KUKA KRL program: MyProgram_041().src

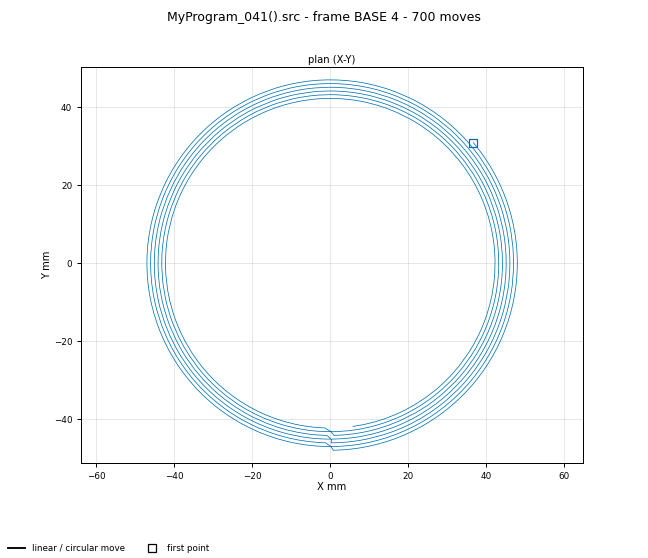
[picture p0: tool path of MyProgram_041().src in frame BASE 4, 700 of 700 moves have a stored position in this frame; points joined in program order, loops and branches not executed]
&ACCESS RVP
&REL 1
&PARAM TEMPLATE = C:\KRC\Roboter\Template\vorgabe
&PARAM EDITMASK = *
DEF MyProgram_041()
; ---- Setting reference (Base) ----
$BASE = BASE_DATA[4]

; --------------------------
; ---- Setting tool (TCP) ----
$TOOL = TOOL_DATA[3]
; --------------------------

$VEL.CP = VEL_APROX_PRINT
Startdeposition()
$VEL.CP = VEL_PRINT
LIN {X 36.6763,Y 30.8604,Z 63,A 32.6646,B 24.8495,C -2.8306,E1 25.1236,E2 -309.1779} C_DIS
LIN {X 38.1464,Y 29.0236,Z 63,A 29.8672,B 24.8502,C -2.8243,E1 25.1284,E2 -306.3787} C_DIS
LIN {X 39.5245,Y 27.1169,Z 63,A 27.0703,B 24.8509,C -2.8177,E1 25.1329,E2 -303.5798} C_DIS
LIN {X 40.8075,Y 25.1448,Z 63,A 24.2742,B 24.8516,C -2.8108,E1 25.1371,E2 -300.7815} C_DIS
LIN {X 41.9921,Y 23.1122,Z 63,A 21.4787,B 24.8523,C -2.8037,E1 25.141,E2 -297.9837} C_DIS
LIN {X 43.0756,Y 21.0239,Z 63,A 18.6835,B 24.8531,C -2.7964,E1 25.1445,E2 -295.1861} C_DIS
LIN {X 44.0553,Y 18.885,Z 63,A 15.8888,B 24.8539,C -2.7889,E1 25.1476,E2 -292.389} C_DIS
LIN {X 44.9289,Y 16.7005,Z 63,A 13.0946,B 24.8547,C -2.7812,E1 25.1505,E2 -289.5921} C_DIS
LIN {X 45.6942,Y 14.4759,Z 63,A 10.3007,B 24.8555,C -2.7734,E1 25.1529,E2 -286.7955} C_DIS
LIN {X 46.3495,Y 12.2163,Z 63,A 7.5073,B 24.8564,C -2.7654,E1 25.155,E2 -283.9992} C_DIS
LIN {X 46.8931,Y 9.9273,Z 63,A 4.7141,B 24.8572,C -2.7573,E1 25.1567,E2 -281.203} C_DIS
LIN {X 47.3237,Y 7.6144,Z 63,A 1.9212,B 24.8581,C -2.749,E1 25.158,E2 -278.4069} C_DIS
LIN {X 47.6194,Y 5.4623,Z 63,A -0.6575,B 24.8589,C -2.7414,E1 25.1589,E2 -275.8254} C_DIS
LIN {X 47.83,Y 3.1192,Z 63,A -3.4502,B 24.8597,C -2.733,E1 25.1596,E2 -273.0294} C_DIS
LIN {X 47.9255,Y 0.7685,Z 63,A -6.2425,B 24.8606,C -2.7246,E1 25.1598,E2 -270.2338} C_DIS
LIN {X 47.9207,Y -1.0254,Z 63,A -8.406,B 24.8613,C -2.7174,E1 25.1597,E2 -268.0664} C_DIS
LIN {X 47.8025,Y -3.5261,Z 63,A -11.3432,B 24.8622,C -2.7091,E1 25.1592,E2 -265.1268} C_DIS
LIN {X 47.5719,Y -5.8674,Z 63,A -14.1356,B 24.863,C -2.7006,E1 25.1583,E2 -262.3309} C_DIS
LIN {X 47.2267,Y -8.1946,Z 63,A -16.9281,B 24.8639,C -2.6922,E1 25.1571,E2 -259.5348} C_DIS
LIN {X 46.7677,Y -10.502,Z 63,A -19.7204,B 24.8647,C -2.6838,E1 25.1555,E2 -256.7389} C_DIS
LIN {X 46.1961,Y -12.7842,Z 63,A -22.5132,B 24.8656,C -2.6755,E1 25.1535,E2 -253.9426} C_DIS
LIN {X 45.5132,Y -15.0355,Z 63,A -25.3061,B 24.8664,C -2.6672,E1 25.1511,E2 -251.146} C_DIS
LIN {X 44.7206,Y -17.2506,Z 63,A -28.0993,B 24.8672,C -2.6591,E1 25.1484,E2 -248.3492} C_DIS
LIN {X 43.8203,Y -19.4242,Z 63,A -30.8927,B 24.868,C -2.6511,E1 25.1454,E2 -245.5521} C_DIS
LIN {X 42.8144,Y -21.5509,Z 63,A -33.6867,B 24.8688,C -2.6432,E1 25.1419,E2 -242.7545} C_DIS
LIN {X 41.7053,Y -23.6258,Z 63,A -36.4807,B 24.8696,C -2.6355,E1 25.1382,E2 -239.957} C_DIS
LIN {X 40.4959,Y -25.6437,Z 63,A -39.2754,B 24.8703,C -2.628,E1 25.1341,E2 -237.1587} C_DIS
LIN {X 39.1888,Y -27.5999,Z 63,A -42.0705,B 24.871,C -2.6207,E1 25.1296,E2 -234.36} C_DIS
LIN {X 37.7873,Y -29.4895,Z 63,A -44.8661,B 24.8717,C -2.6136,E1 25.1249,E2 -231.5609} C_DIS
LIN {X 36.2948,Y -31.3081,Z 63,A -47.6623,B 24.8724,C -2.6067,E1 25.1199,E2 -228.7612} C_DIS
LIN {X 34.7149,Y -33.0513,Z 63,A -50.4591,B 24.8731,C -2.6001,E1 25.1146,E2 -225.961} C_DIS
LIN {X 32.9356,Y -34.8237,Z 63,A -53.4601,B 24.8738,C -2.5931,E1 25.1086,E2 -222.9559} C_DIS
LIN {X 31.0875,Y -36.4828,Z 63,A -56.467,B 24.8745,C -2.5857,E1 25.1022,E2 -219.9435} C_DIS
LIN {X 29.0236,Y -38.1464,Z 63,A -59.5531,B 24.875,C -2.5805,E1 25.0954,E2 -216.8565} C_DIS
LIN {X 27.1169,Y -39.5245,Z 63,A -62.3528,B 24.8755,C -2.5751,E1 25.089,E2 -214.0537} C_DIS
LIN {X 25.1448,Y -40.8075,Z 63,A -65.1533,B 24.876,C -2.5701,E1 25.0824,E2 -211.2502} C_DIS
LIN {X 23.1122,Y -41.9921,Z 63,A -67.9546,B 24.8765,C -2.5654,E1 25.0756,E2 -208.4461} C_DIS
LIN {X 21.0239,Y -43.0756,Z 63,A -70.7565,B 24.8769,C -2.561,E1 25.0686,E2 -205.6414} C_DIS
LIN {X 18.885,Y -44.0553,Z 63,A -73.5596,B 24.8773,C -2.557,E1 25.0615,E2 -202.8357} C_DIS
LIN {X 16.7005,Y -44.9289,Z 63,A -76.3635,B 24.8776,C -2.5534,E1 25.0542,E2 -200.0294} C_DIS
LIN {X 14.4759,Y -45.6942,Z 63,A -79.1682,B 24.8779,C -2.5501,E1 25.0467,E2 -197.2223} C_DIS
LIN {X 12.2163,Y -46.3495,Z 63,A -81.9739,B 24.8782,C -2.5472,E1 25.0392,E2 -194.4144} C_DIS
LIN {X 9.9273,Y -46.8931,Z 63,A -84.7806,B 24.8784,C -2.5448,E1 25.0315,E2 -191.6057} C_DIS
LIN {X 7.6145,Y -47.3237,Z 63,A -87.5882,B 24.8786,C -2.5427,E1 25.0238,E2 -188.7961} C_DIS
LIN {X 5.4623,Y -47.6194,Z 63,A -90.0984,B 24.8786,C -2.5426,E1 25.0168,E2 -186.2875} C_DIS
LIN {X 3.1192,Y -47.83,Z 63,A -92.991,B 24.8789,C -2.5399,E1 25.0088,E2 -183.3901} C_DIS
LIN {X 0.7685,Y -47.9255,Z 63,A -95.7979,B 24.8789,C -2.5391,E1 25.0009,E2 -180.5818} C_DIS
LIN {X 0.7685,Y -47.9255,Z 63,A -95.7979,B 24.8789,C -2.5391,E1 25.0009,E2 -180.5818} C_DIS
Enddeposition()
LIN {X 0.2143,Y -46.9784,Z 63,A -95.4397,B 24.8758,C -2.5723,E1 25.0021,E2 -181.019} C_DIS
Startdeposition()
$VEL.CP = VEL_PRINT
LIN {X 2.5559,Y -46.9121,Z 63,A -92.1955,B 24.8751,C -2.5797,E1 25.0112,E2 -184.2799} C_DIS
LIN {X 5.1846,Y -46.6955,Z 63,A -89.0891,B 24.8751,C -2.5796,E1 25.0199,E2 -187.3841} C_DIS
LIN {X 7.4092,Y -46.3943,Z 63,A -86.2366,B 24.8747,C -2.5834,E1 25.0278,E2 -190.2431} C_DIS
LIN {X 9.682,Y -45.9738,Z 63,A -83.5774,B 24.8747,C -2.583,E1 25.035,E2 -192.8981} C_DIS
LIN {X 12.0789,Y -45.4027,Z 63,A -80.419,B 24.8742,C -2.5887,E1 25.0436,E2 -196.0652} C_DIS
LIN {X 14.5681,Y -44.6661,Z 63,A -77.3449,B 24.874,C -2.5907,E1 25.0518,E2 -199.1385} C_DIS
LIN {X 16.8661,Y -43.8505,Z 63,A -74.3809,B 24.8736,C -2.5944,E1 25.0596,E2 -202.105} C_DIS
LIN {X 19.0655,Y -42.94,Z 63,A -71.3711,B 24.873,C -2.6005,E1 25.0673,E2 -205.1221} C_DIS
LIN {X 21.5139,Y -41.7666,Z 63,A -68.1734,B 24.8727,C -2.6038,E1 25.0753,E2 -208.319} C_DIS
LIN {X 23.5958,Y -40.6271,Z 63,A -65.3023,B 24.8723,C -2.6084,E1 25.0823,E2 -211.1926} C_DIS
LIN {X 25.6235,Y -39.3801,Z 63,A -62.7798,B 24.8724,C -2.6069,E1 25.0882,E2 -213.7033} C_DIS
LIN {X 27.3032,Y -38.2334,Z 63,A -59.8844,B 24.8712,C -2.6194,E1 25.0949,E2 -216.6186} C_DIS
LIN {X 29.4691,Y -36.5899,Z 63,A -56.4143,B 24.8702,C -2.6293,E1 25.1026,E2 -220.0991} C_DIS
LIN {X 31.6335,Y -34.7366,Z 63,A -52.8319,B 24.8692,C -2.6391,E1 25.1101,E2 -223.6906} C_DIS
LIN {X 33.711,Y -32.7242,Z 63,A -49.5665,B 24.8689,C -2.6426,E1 25.1165,E2 -226.9504} C_DIS
LIN {X 35.4262,Y -30.8588,Z 63,A -46.5387,B 24.8682,C -2.6491,E1 25.1221,E2 -229.9802} C_DIS
LIN {X 36.9362,Y -29.0346,Z 63,A -43.7525,B 24.8677,C -2.6547,E1 25.127,E2 -232.7665} C_DIS
LIN {X 38.153,Y -27.4162,Z 63,A -41.5295,B 24.8675,C -2.6566,E1 25.1307,E2 -234.9833} C_DIS
LIN {X 39.4006,Y -25.5917,Z 63,A -38.491,B 24.8661,C -2.6705,E1 25.1354,E2 -238.0396} C_DIS
LIN {X 40.6723,Y -23.5171,Z 63,A -35.6061,B 24.8654,C -2.6773,E1 25.1395,E2 -240.9257} C_DIS
LIN {X 41.8533,Y -21.3443,Z 63,A -32.6333,B 24.8646,C -2.6851,E1 25.1434,E2 -243.9014} C_DIS
LIN {X 42.6017,Y -19.8084,Z 63,A -30.3873,B 24.8637,C -2.6944,E1 25.146,E2 -246.1573} C_DIS
LIN {X 43.7378,Y -17.1547,Z 63,A -27.0571,B 24.863,C -2.7012,E1 25.1496,E2 -249.4853} C_DIS
LIN {X 44.6118,Y -14.7336,Z 63,A -23.7996,B 24.8618,C -2.7131,E1 25.1525,E2 -252.7525} C_DIS
LIN {X 45.4336,Y -11.9641,Z 63,A -20.8446,B 24.8618,C -2.7129,E1 25.1548,E2 -255.6901} C_DIS
LIN {X 46.1112,Y -9.0029,Z 63,A -15.9869,B 24.8583,C -2.747,E1 25.1576,E2 -260.6001} C_DIS
LIN {X 46.6067,Y -5.9251,Z 63,A -12.4483,B 24.8576,C -2.7537,E1 25.1589,E2 -264.1337} C_DIS
LIN {X 46.9567,Y -1.5325,Z 63,A -7.5964,B 24.8569,C -2.7604,E1 25.1598,E2 -268.9726} C_DIS
LIN {X 46.9771,Y 0.6801,Z 63,A -4.6126,B 24.8554,C -2.7744,E1 25.1597,E2 -271.9719} C_DIS
LIN {X 46.8023,Y 4.1062,Z 63,A -0.522,B 24.8542,C -2.7856,E1 25.1589,E2 -276.0648} C_DIS
LIN {X 46.3299,Y 7.7988,Z 63,A 3.3596,B 24.8542,C -2.7869,E1 25.1574,E2 -279.9263} C_DIS
LIN {X 45.9041,Y 10.0043,Z 63,A 6.6583,B 24.8521,C -2.806,E1 25.1555,E2 -283.251} C_DIS
LIN {X 45.2529,Y 12.6287,Z 63,A 9.5452,B 24.8519,C -2.8079,E1 25.1534,E2 -286.1258} C_DIS
LIN {X 44.6509,Y 14.615,Z 63,A 12.1852,B 24.8509,C -2.8174,E1 25.1512,E2 -288.7733} C_DIS
LIN {X 43.8399,Y 16.8942,Z 63,A 15.8973,B 24.8484,C -2.8405,E1 25.1475,E2 -292.5194} C_DIS
LIN {X 42.3575,Y 20.3254,Z 63,A 19.7008,B 24.8486,C -2.8387,E1 25.1431,E2 -296.298} C_DIS
LIN {X 41.1665,Y 22.6422,Z 63,A 22.7618,B 24.8479,C -2.8449,E1 25.1391,E2 -299.3577} C_DIS
LIN {X 40.0354,Y 24.5864,Z 63,A 25.8315,B 24.8465,C -2.8582,E1 25.1347,E2 -302.4431} C_DIS
LIN {X 38.3506,Y 27.1393,Z 63,A 29.1136,B 24.8465,C -2.859,E1 25.1295,E2 -305.7111} C_DIS
LIN {X 37.1165,Y 28.8039,Z 63,A 31.388,B 24.8463,C -2.8604,E1 25.1257,E2 -307.9778} C_DIS
LIN {X 35.589,Y 30.672,Z 63,A 34.6406,B 24.8449,C -2.8728,E1 25.1199,E2 -311.2449} C_DIS
LIN {X 34.078,Y 32.3421,Z 63,A 37.4842,B 24.8441,C -2.8805,E1 25.1145,E2 -314.0943} C_DIS
LIN {X 32.1994,Y 34.2122,Z 63,A 40.6791,B 24.8435,C -2.8864,E1 25.108,E2 -317.2899} C_DIS
LIN {X 30.3202,Y 35.8887,Z 63,A 43.688,B 24.8429,C -2.8911,E1 25.1017,E2 -320.2982} C_DIS
LIN {X 28.4537,Y 37.3863,Z 63,A 46.7319,B 24.8421,C -2.8986,E1 25.095,E2 -323.3484} C_DIS
LIN {X 26.3,Y 38.9303,Z 63,A 49.9644,B 24.8416,C -2.9038,E1 25.0876,E2 -326.5823} C_DIS
LIN {X 23.9042,Y 40.4458,Z 63,A 53.0971,B 24.8416,C -2.9032,E1 25.0801,E2 -329.7037} C_DIS
LIN {X 21.9009,Y 41.5647,Z 63,A 56.1163,B 24.8408,C -2.9108,E1 25.0727,E2 -332.7322} C_DIS
LIN {X 20.3598,Y 42.3409,Z 63,A 58.9872,B 24.8391,C -2.9266,E1 25.0654,E2 -335.6331} C_DIS
LIN {X 16.672,Y 43.924,Z 63,A 63.0887,B 24.84,C -2.9178,E1 25.0549,E2 -339.7044} C_DIS
LIN {X 14.163,Y 44.7968,Z 63,A 66.3896,B 24.8396,C -2.9214,E1 25.0461,E2 -343.0076} C_DIS
LIN {X 11.5862,Y 45.5307,Z 63,A 69.5926,B 24.8396,C -2.9224,E1 25.0375,E2 -346.2078} C_DIS
LIN {X 8.9483,Y 46.1217,Z 63,A 72.8147,B 24.8395,C -2.9226,E1 25.0287,E2 -349.4264} C_DIS
LIN {X 7.0373,Y 46.4518,Z 63,A 75.1648,B 24.8395,C -2.9231,E1 25.0222,E2 -351.7753} C_DIS
LIN {X 4.6739,Y 46.7491,Z 63,A 78.1637,B 24.8392,C -2.9251,E1 25.0139,E2 -354.7767} C_DIS
LIN {X 2.015,Y 46.9384,Z 63,A 81.4087,B 24.8392,C -2.9249,E1 25.0048,E2 -358.0203} C_DIS
LIN {X -0.6275,Y 46.9781,Z 63,A 84.1397,B 24.8402,C -2.9165,E1 24.9973,E2 -360.7311} C_DIS
LIN {X -2.9749,Y 46.8878,Z 63,A 87.5384,B 24.8393,C -2.9239,E1 24.9877,E2 -364.1482} C_DIS
LIN {X -5.5799,Y 46.6493,Z 63,A 90.7209,B 24.8395,C -2.9221,E1 24.9789,E2 -367.3283} C_DIS
LIN {X -7.976,Y 46.3002,Z 63,A 93.578,B 24.8399,C -2.9186,E1 24.971,E2 -370.1797} C_DIS
LIN {X -10.1804,Y 45.8657,Z 63,A 96.0614,B 24.8406,C -2.9125,E1 24.9643,E2 -372.6513} C_DIS
LIN {X -12.438,Y 45.3057,Z 63,A 99.2139,B 24.8404,C -2.9144,E1 24.9557,E2 -375.8132} C_DIS
LIN {X -14.0781,Y 44.8231,Z 63,A 102.2726,B 24.839,C -2.9267,E1 24.9475,E2 -378.9066} C_DIS
LIN {X -17.8756,Y 43.4484,Z 63,A 106.2167,B 24.8414,C -2.9057,E1 24.9373,E2 -382.8088} C_DIS
LIN {X -20.1909,Y 42.4221,Z 63,A 109.3156,B 24.8418,C -2.9012,E1 24.9295,E2 -385.9049} C_DIS
LIN {X -21.88,Y 41.5757,Z 63,A 112.0704,B 24.8415,C -2.904,E1 24.9226,E2 -388.6739} C_DIS
LIN {X -24.7808,Y 39.915,Z 63,A 115.744,B 24.843,C -2.891,E1 24.9139,E2 -392.3276} C_DIS
LIN {X -26.8595,Y 38.5467,Z 63,A 118.8267,B 24.8435,C -2.8858,E1 24.9068,E2 -395.4084} C_DIS
LIN {X -29.0273,Y 36.9419,Z 63,A 122.1517,B 24.8442,C -2.8796,E1 24.8994,E2 -398.7304} C_DIS
LIN {X -31.0833,Y 35.2301,Z 63,A 124.9609,B 24.8457,C -2.8662,E1 24.8935,E2 -401.5186} C_DIS
LIN {X -32.2942,Y 34.123,Z 63,A 127.5606,B 24.8453,C -2.8698,E1 24.8881,E2 -404.1375} C_DIS
LIN {X -34.3301,Y 32.074,Z 63,A 130.986,B 24.8463,C -2.8601,E1 24.8815,E2 -407.5544} C_DIS
LIN {X -36.1116,Y 30.0538,Z 63,A 134.2654,B 24.8472,C -2.8518,E1 24.8755,E2 -410.8289} C_DIS
LIN {X -37.7375,Y 27.9862,Z 63,A 137.0526,B 24.8487,C -2.8378,E1 24.8708,E2 -413.5958} C_DIS
LIN {X -38.8546,Y 26.4122,Z 63,A 139.9102,B 24.8487,C -2.8382,E1 24.8663,E2 -416.4685} C_DIS
LIN {X -40.3999,Y 23.982,Z 63,A 143.4333,B 24.8497,C -2.8286,E1 24.8611,E2 -419.9866} C_DIS
LIN {X -41.7299,Y 21.5857,Z 63,A 146.753,B 24.8507,C -2.8187,E1 24.8567,E2 -423.3003} C_DIS
LIN {X -42.7838,Y 19.4124,Z 63,A 149.9969,B 24.8512,C -2.814,E1 24.8529,E2 -426.5507} C_DIS
LIN {X -44.1351,Y 16.1049,Z 63,A 154.0955,B 24.853,C -2.7976,E1 24.8488,E2 -430.633} C_DIS
LIN {X -44.8607,Y 13.9568,Z 63,A 156.6924,B 24.8541,C -2.787,E1 24.8466,E2 -433.2194} C_DIS
LIN {X -45.5111,Y 11.6624,Z 63,A 159.7162,B 24.8549,C -2.7795,E1 24.8443,E2 -436.2429} C_DIS
LIN {X -46.0396,Y 9.3616,Z 63,A 162.7323,B 24.8556,C -2.7723,E1 24.8426,E2 -439.2596} C_DIS
LIN {X -46.4956,Y 6.7422,Z 63,A 165.7745,B 24.857,C -2.7596,E1 24.8412,E2 -442.2894} C_DIS
LIN {X -46.7606,Y 4.558,Z 63,A 168.776,B 24.8574,C -2.7553,E1 24.8403,E2 -445.2986} C_DIS
LIN {X -46.9449,Y 1.8632,Z 63,A 171.9898,B 24.8586,C -2.7439,E1 24.8398,E2 -448.5045} C_DIS
LIN {X -46.9769,Y -0.6903,Z 63,A 175.163,B 24.8595,C -2.7349,E1 24.8398,E2 -451.6753} C_DIS
LIN {X -46.8667,Y -3.2866,Z 63,A 178.2443,B 24.8607,C -2.7239,E1 24.8403,E2 -454.7488} C_DIS
LIN {X -46.6945,Y -5.1937,Z 63,A -179.2053,B 24.8611,C -2.7194,E1 24.8411,E2 -457.3038} C_DIS
LIN {X -46.3138,Y -7.8948,Z 63,A -175.9746,B 24.8623,C -2.708,E1 24.8425,E2 -460.5264} C_DIS
LIN {X -45.8138,Y -10.4116,Z 63,A -172.7879,B 24.8632,C -2.6993,E1 24.8443,E2 -463.711} C_DIS
LIN {X -45.1647,Y -12.9399,Z 63,A -169.5411,B 24.864,C -2.6907,E1 24.8467,E2 -466.9561} C_DIS
LIN {X -44.3842,Y -15.4059,Z 63,A -166.7067,B 24.8654,C -2.6773,E1 24.8492,E2 -469.7745} C_DIS
LIN {X -43.6542,Y -17.3676,Z 63,A -163.9593,B 24.8659,C -2.6726,E1 24.8519,E2 -472.5262} C_DIS
LIN {X -42.5994,Y -19.8133,Z 63,A -160.4602,B 24.8664,C -2.6669,E1 24.8559,E2 -476.031} C_DIS
LIN {X -41.346,Y -22.3113,Z 63,A -157.1221,B 24.8675,C -2.6568,E1 24.8602,E2 -479.3628} C_DIS
LIN {X -40.0037,Y -24.6386,Z 63,A -153.944,B 24.8684,C -2.647,E1 24.8647,E2 -482.5338} C_DIS
LIN {X -38.8415,Y -26.4316,Z 63,A -151.505,B 24.8693,C -2.6382,E1 24.8685,E2 -484.9641} C_DIS
LIN {X -37.5666,Y -28.2139,Z 63,A -148.5222,B 24.8695,C -2.6361,E1 24.8734,E2 -487.9563} C_DIS
LIN {X -35.9165,Y -30.2876,Z 63,A -145.3045,B 24.8703,C -2.6285,E1 24.8791,E2 -491.1707} C_DIS
LIN {X -34.1655,Y -32.249,Z 63,A -142.6079,B 24.8717,C -2.6144,E1 24.8842,E2 -493.8456} C_DIS
LIN {X -32.5987,Y -33.832,Z 63,A -139.3792,B 24.8715,C -2.6161,E1 24.8906,E2 -497.0918} C_DIS
LIN {X -30.6979,Y -35.5667,Z 63,A -136.1305,B 24.8719,C -2.6116,E1 24.8974,E2 -500.3429} C_DIS
LIN {X -29.145,Y -36.8489,Z 63,A -133.9522,B 24.8728,C -2.6032,E1 24.9021,E2 -502.5092} C_DIS
LIN {X -27.314,Y -38.2259,Z 63,A -130.9734,B 24.873,C -2.6012,E1 24.9088,E2 -505.4939} C_DIS
LIN {X -25.1237,Y -39.6996,Z 63,A -127.4866,B 24.873,C -2.6003,E1 24.917,E2 -508.9897} C_DIS
LIN {X -22.9515,Y -40.994,Z 63,A -124.3564,B 24.8734,C -2.5968,E1 24.9246,E2 -512.1208} C_DIS
LIN {X -20.2336,Y -42.4016,Z 63,A -120.8547,B 24.8742,C -2.5888,E1 24.9333,E2 -515.6127} C_DIS
LIN {X -18.3269,Y -43.2598,Z 63,A -118.4196,B 24.8746,C -2.5844,E1 24.9395,E2 -518.043} C_DIS
LIN {X -16.0279,Y -44.1632,Z 63,A -115.2725,B 24.8746,C -2.5837,E1 24.9478,E2 -521.1952} C_DIS
LIN {X -13.4838,Y -45.0053,Z 63,A -111.9643,B 24.8748,C -2.582,E1 24.9566,E2 -524.5051} C_DIS
LIN {X -10.8546,Y -45.7114,Z 63,A -108.855,B 24.8753,C -2.5768,E1 24.965,E2 -527.6066} C_DIS
LIN {X -8.6723,Y -46.1748,Z 63,A -106.0396,B 24.8753,C -2.5773,E1 24.9727,E2 -530.4262} C_DIS
LIN {X -6.3616,Y -46.5496,Z 63,A -103.1497,B 24.8753,C -2.5772,E1 24.9807,E2 -533.3183} C_DIS
LIN {X -3.8273,Y -46.8256,Z 63,A -99.9519,B 24.8752,C -2.5784,E1 24.9896,E2 -536.5206} C_DIS
LIN {X -1.3952,Y -46.961,Z 63,A -97.0343,B 24.8752,C -2.5778,E1 24.9977,E2 -539.4375} C_DIS
LIN {X 0.2143,Y -46.9784,Z 63,A -95.4395,B 24.8758,C -2.5722,E1 25.0021,E2 -541.019} C_DIS
Enddeposition()
LIN {X 0.2143,Y -46.9784,Z 63,A -95.4395,B 24.8758,C -2.5722,E1 25.0021,E2 -541.019} C_DIS
Startdeposition()
$VEL.CP = VEL_PRINT
LIN {X -1.2064,Y -46.0165,Z 63,A -98.1296,B 24.8757,C -2.5734,E1 24.9946,E2 -538.3316} C_DIS
LIN {X -2.996,Y -45.9343,Z 63,A -100.6273,B 24.8761,C -2.5691,E1 24.9876,E2 -535.823} C_DIS
LIN {X -5.5683,Y -45.6943,Z 63,A -103.8573,B 24.8761,C -2.5693,E1 24.9787,E2 -532.5914} C_DIS
LIN {X -8.1693,Y -45.3011,Z 63,A -107.3449,B 24.8763,C -2.567,E1 24.969,E2 -529.0951} C_DIS
LIN {X -10.6177,Y -44.7912,Z 63,A -110.1372,B 24.8757,C -2.5732,E1 24.9615,E2 -526.314} C_DIS
LIN {X -12.9468,Y -44.1739,Z 63,A -113.2311,B 24.8757,C -2.5737,E1 24.9531,E2 -523.2164} C_DIS
LIN {X -15.3538,Y -43.3959,Z 63,A -116.3054,B 24.8753,C -2.5773,E1 24.945,E2 -520.1448} C_DIS
LIN {X -18.1446,Y -42.3057,Z 63,A -119.8982,B 24.8748,C -2.5829,E1 24.9357,E2 -516.5574} C_DIS
LIN {X -19.9975,Y -41.4612,Z 63,A -122.8081,B 24.875,C -2.5804,E1 24.9283,E2 -513.6341} C_DIS
LIN {X -22.5947,Y -40.1054,Z 63,A -125.9036,B 24.8738,C -2.5929,E1 24.9208,E2 -510.5598} C_DIS
LIN {X -23.9436,Y -39.3146,Z 63,A -128.1392,B 24.8739,C -2.5916,E1 24.9154,E2 -508.3143} C_DIS
LIN {X -25.6481,Y -38.2249,Z 63,A -130.5652,B 24.8734,C -2.5967,E1 24.9097,E2 -505.8925} C_DIS
LIN {X -27.056,Y -37.2411,Z 63,A -133.252,B 24.8738,C -2.5926,E1 24.9036,E2 -503.1867} C_DIS
LIN {X -28.9064,Y -35.824,Z 63,A -135.8534,B 24.8729,C -2.6019,E1 24.8979,E2 -500.5977} C_DIS
LIN {X -30.8319,Y -34.1812,Z 63,A -138.9812,B 24.8723,C -2.6082,E1 24.8914,E2 -497.4727} C_DIS
LIN {X -33.3178,Y -31.7629,Z 63,A -142.8699,B 24.8708,C -2.6228,E1 24.8837,E2 -493.6024} C_DIS
LIN {X -35.1938,Y -29.6705,Z 63,A -146.9276,B 24.8708,C -2.6231,E1 24.8762,E2 -489.5271} C_DIS
LIN {X -36.5981,Y -27.9205,Z 63,A -149.5235,B 24.8699,C -2.6322,E1 24.8717,E2 -486.9408} C_DIS
LIN {X -38.1584,Y -25.7462,Z 63,A -152.927,B 24.8692,C -2.6394,E1 24.8663,E2 -483.5377} C_DIS
LIN {X -39.398,Y -23.8063,Z 63,A -155.8746,B 24.8686,C -2.6456,E1 24.8619,E2 -480.5899} C_DIS
LIN {X -40.6461,Y -21.6068,Z 63,A -159.8006,B 24.8687,C -2.6441,E1 24.8567,E2 -476.6397} C_DIS
LIN {X -41.8492,Y -19.1742,Z 63,A -163.1919,B 24.8678,C -2.6532,E1 24.8527,E2 -473.2516} C_DIS
LIN {X -43.1775,Y -15.9583,Z 63,A -166.9255,B 24.8658,C -2.673,E1 24.8489,E2 -469.5443} C_DIS
LIN {X -44.4043,Y -12.1328,Z 63,A -171.4229,B 24.8637,C -2.6939,E1 24.8453,E2 -465.0712} C_DIS
LIN {X -44.8415,Y -10.4003,Z 63,A -174.104,B 24.8637,C -2.6949,E1 24.8435,E2 -462.3767} C_DIS
LIN {X -45.347,Y -7.9143,Z 63,A -177.23,B 24.8626,C -2.7049,E1 24.8418,E2 -459.2561} C_DIS
LIN {X -45.7486,Y -5.1043,Z 63,A 178.9324,B 24.8619,C -2.7121,E1 24.8405,E2 -455.4127} C_DIS
LIN {X -45.971,Y -2.3719,Z 63,A 175.7437,B 24.8605,C -2.7254,E1 24.8399,E2 -452.2368} C_DIS
LIN {X -46.0317,Y 0.1331,Z 63,A 172.5788,B 24.8595,C -2.7346,E1 24.8398,E2 -449.0748} C_DIS
LIN {X -45.9564,Y 2.6362,Z 63,A 169.1185,B 24.859,C -2.7403,E1 24.8402,E2 -445.6072} C_DIS
LIN {X -45.6948,Y 5.5633,Z 63,A 165.7078,B 24.8575,C -2.7547,E1 24.8412,E2 -442.2107} C_DIS
LIN {X -45.3131,Y 8.1024,Z 63,A 162.5598,B 24.8564,C -2.7653,E1 24.8427,E2 -439.0693} C_DIS
LIN {X -44.8166,Y 10.5083,Z 63,A 159.1164,B 24.8559,C -2.7701,E1 24.8448,E2 -435.6172} C_DIS
LIN {X -43.7953,Y 14.1738,Z 63,A 154.9462,B 24.8536,C -2.7916,E1 24.848,E2 -431.4741} C_DIS
LIN {X -42.8735,Y 16.7571,Z 63,A 151.1618,B 24.853,C -2.7973,E1 24.8517,E2 -427.682} C_DIS
LIN {X -42.0147,Y 18.8062,Z 63,A 148.3926,B 24.8522,C -2.8054,E1 24.8548,E2 -424.917} C_DIS
LIN {X -40.6841,Y 21.5346,Z 63,A 144.617,B 24.851,C -2.8163,E1 24.8595,E2 -421.1473} C_DIS
LIN {X -39.3588,Y 23.8709,Z 63,A 141.6249,B 24.8495,C -2.8301,E1 24.8637,E2 -418.1726} C_DIS
LIN {X -38.6201,Y 25.0484,Z 63,A 139.4394,B 24.8496,C -2.8291,E1 24.867,E2 -415.9737} C_DIS
LIN {X -36.9044,Y 27.514,Z 63,A 135.8359,B 24.8484,C -2.8408,E1 24.8729,E2 -412.3806} C_DIS
LIN {X -35.4039,Y 29.4193,Z 63,A 132.7229,B 24.8477,C -2.8473,E1 24.8783,E2 -409.2687} C_DIS
LIN {X -33.7426,Y 31.3119,Z 63,A 129.389,B 24.8471,C -2.8525,E1 24.8846,E2 -405.9323} C_DIS
LIN {X -31.9643,Y 33.1242,Z 63,A 126.5284,B 24.8459,C -2.8638,E1 24.8902,E2 -403.0866} C_DIS
LIN {X -30.202,Y 34.7387,Z 63,A 123.6989,B 24.845,C -2.8723,E1 24.8961,E2 -400.2662} C_DIS
LIN {X -28.6374,Y 36.0394,Z 63,A 120.8381,B 24.8449,C -2.8734,E1 24.9023,E2 -397.3972} C_DIS
LIN {X -26.6472,Y 37.5349,Z 63,A 117.7975,B 24.8441,C -2.8804,E1 24.9091,E2 -394.3625} C_DIS
LIN {X -24.4411,Y 39.0073,Z 63,A 114.7548,B 24.8431,C -2.8901,E1 24.9162,E2 -391.333} C_DIS
LIN {X -22.3162,Y 40.2609,Z 63,A 110.9738,B 24.8435,C -2.8857,E1 24.9254,E2 -387.5306} C_DIS
LIN {X -20.0871,Y 41.4182,Z 63,A 107.6112,B 24.8434,C -2.8874,E1 24.9339,E2 -384.1632} C_DIS
LIN {X -16.1624,Y 43.1014,Z 63,A 103.0742,B 24.8414,C -2.9054,E1 24.9455,E2 -379.659} C_DIS
LIN {X -14.2429,Y 43.773,Z 63,A 100.4956,B 24.8411,C -2.9078,E1 24.9523,E2 -377.0811} C_DIS
LIN {X -10.1995,Y 44.8879,Z 63,A 95.3599,B 24.8404,C -2.9142,E1 24.9662,E2 -371.953} C_DIS
LIN {X -8.1604,Y 45.3027,Z 63,A 92.5223,B 24.8406,C -2.9126,E1 24.974,E2 -369.1086} C_DIS
LIN {X -5.6136,Y 45.689,Z 63,A 89.3437,B 24.8403,C -2.915,E1 24.9828,E2 -365.9331} C_DIS
LIN {X -2.5568,Y 45.9608,Z 63,A 85.1701,B 24.8407,C -2.9113,E1 24.9944,E2 -361.7493} C_DIS
LIN {X 0.0461,Y 46.0324,Z 63,A 82.2478,B 24.8401,C -2.9169,E1 25.0025,E2 -358.84} C_DIS
LIN {X 2.4996,Y 45.9639,Z 63,A 79.2706,B 24.84,C -2.9183,E1 25.0108,E2 -355.867} C_DIS
LIN {X 4.9421,Y 45.766,Z 63,A 75.7328,B 24.8408,C -2.9104,E1 25.0207,E2 -352.3127} C_DIS
LIN {X 7.7136,Y 45.3811,Z 63,A 72.8041,B 24.84,C -2.9181,E1 25.0287,E2 -349.405} C_DIS
LIN {X 10.0408,Y 44.924,Z 63,A 69.7888,B 24.8403,C -2.9157,E1 25.037,E2 -346.3879} C_DIS
LIN {X 12.1877,Y 44.3894,Z 63,A 66.9591,B 24.8406,C -2.9128,E1 25.0446,E2 -343.5558} C_DIS
LIN {X 15.2052,Y 43.448,Z 63,A 63.4061,B 24.8402,C -2.916,E1 25.054,E2 -340.0168} C_DIS
LIN {X 16.9863,Y 42.7834,Z 63,A 60.0201,B 24.8423,C -2.8971,E1 25.0629,E2 -336.5935} C_DIS
LIN {X 19.9698,Y 41.4745,Z 63,A 56.8434,B 24.8412,C -2.9069,E1 25.0709,E2 -333.4482} C_DIS
LIN {X 22.0641,Y 40.3995,Z 63,A 53.6806,B 24.8421,C -2.8993,E1 25.0787,E2 -330.2761} C_DIS
LIN {X 24.0663,Y 39.24,Z 63,A 50.9303,B 24.8423,C -2.8973,E1 25.0853,E2 -327.5297} C_DIS
LIN {X 26.2362,Y 37.8232,Z 63,A 48.1435,B 24.842,C -2.8997,E1 25.0918,E2 -324.7579} C_DIS
LIN {X 27.6646,Y 36.7913,Z 63,A 45.3701,B 24.8435,C -2.8861,E1 25.0981,E2 -321.9618} C_DIS
LIN {X 30.7034,Y 34.2962,Z 63,A 40.7495,B 24.844,C -2.8817,E1 25.1079,E2 -317.3487} C_DIS
LIN {X 32.3072,Y 32.7899,Z 63,A 37.8008,B 24.845,C -2.8724,E1 25.1139,E2 -314.3904} C_DIS
LIN {X 34.1928,Y 30.8189,Z 63,A 34.493,B 24.8456,C -2.8666,E1 25.1202,E2 -311.0833} C_DIS
LIN {X 35.7052,Y 29.053,Z 63,A 31.6081,B 24.8463,C -2.8602,E1 25.1253,E2 -308.1964} C_DIS
LIN {X 36.9867,Y 27.4041,Z 63,A 28.9067,B 24.8472,C -2.8522,E1 25.1299,E2 -305.4888} C_DIS
LIN {X 38.4565,Y 25.2988,Z 63,A 25.491,B 24.8484,C -2.8403,E1 25.1352,E2 -302.0619} C_DIS
LIN {X 40.3477,Y 22.1596,Z 63,A 21.7368,B 24.8481,C -2.843,E1 25.1405,E2 -298.3336} C_DIS
LIN {X 41.4444,Y 20.0322,Z 63,A 18.2749,B 24.85,C -2.8261,E1 25.1449,E2 -294.8501} C_DIS
LIN {X 42.3895,Y 17.9447,Z 63,A 15.3015,B 24.851,C -2.816,E1 25.1482,E2 -291.8689} C_DIS
LIN {X 43.5032,Y 15.0479,Z 63,A 11.6774,B 24.8518,C -2.8092,E1 25.1517,E2 -288.2491} C_DIS
LIN {X 44.2741,Y 12.5988,Z 63,A 8.4945,B 24.8527,C -2.8001,E1 25.1542,E2 -285.0626} C_DIS
LIN {X 45.1951,Y 8.7369,Z 63,A 3.9388,B 24.8535,C -2.7924,E1 25.1571,E2 -280.5151} C_DIS
LIN {X 45.499,Y 6.9835,Z 63,A 1.2847,B 24.8551,C -2.7774,E1 25.1583,E2 -277.8412} C_DIS
LIN {X 45.8293,Y 4.3144,Z 63,A -1.9546,B 24.856,C -2.769,E1 25.1593,E2 -274.6013} C_DIS
LIN {X 45.997,Y 1.7992,Z 63,A -4.8438,B 24.8565,C -2.7639,E1 25.1597,E2 -271.717} C_DIS
LIN {X 46.0324,Y -0.002,Z 63,A -7.0895,B 24.8573,C -2.7568,E1 25.1597,E2 -269.4679} C_DIS
LIN {X 45.9636,Y -2.5055,Z 63,A -10.5295,B 24.8589,C -2.7409,E1 25.1594,E2 -266.011} C_DIS
LIN {X 45.7414,Y -5.1655,Z 63,A -13.4266,B 24.8592,C -2.7384,E1 25.1586,E2 -263.1251} C_DIS
LIN {X 45.5523,Y -6.629,Z 63,A -16.0411,B 24.8612,C -2.7181,E1 25.1576,E2 -260.478} C_DIS
LIN {X 44.7287,Y -10.8752,Z 63,A -20.3104,B 24.8608,C -2.7222,E1 25.1552,E2 -256.2432} C_DIS
LIN {X 44.2866,Y -12.5548,Z 63,A -22.9638,B 24.8625,C -2.7063,E1 25.1532,E2 -253.5675} C_DIS
LIN {X 43.6072,Y -14.7417,Z 63,A -25.7733,B 24.8633,C -2.6984,E1 25.1508,E2 -250.7551} C_DIS
LIN {X 42.8512,Y -16.8137,Z 63,A -28.7048,B 24.8645,C -2.6866,E1 25.1479,E2 -247.8121} C_DIS
LIN {X 41.568,Y -19.7753,Z 63,A -32.5578,B 24.8653,C -2.6778,E1 25.1434,E2 -243.9592} C_DIS
LIN {X 40.445,Y -21.9803,Z 63,A -35.6266,B 24.8662,C -2.6691,E1 25.1394,E2 -240.8861} C_DIS
LIN {X 39.1602,Y -24.1962,Z 63,A -39.3604,B 24.8681,C -2.6502,E1 25.134,E2 -237.1265} C_DIS
LIN {X 37.1129,Y -27.2317,Z 63,A -42.825,B 24.8673,C -2.6579,E1 25.1286,E2 -233.6971} C_DIS
LIN {X 36.0851,Y -28.5797,Z 63,A -45.4159,B 24.8688,C -2.6436,E1 25.1241,E2 -231.0845} C_DIS
LIN {X 34.4626,Y -30.5175,Z 63,A -48.5896,B 24.8696,C -2.6351,E1 25.1183,E2 -227.9052} C_DIS
LIN {X 32.7997,Y -32.2973,Z 63,A -52.576,B 24.872,C -2.6108,E1 25.1104,E2 -223.8782} C_DIS
LIN {X 29.9252,Y -34.9774,Z 63,A -56.6769,B 24.8717,C -2.6137,E1 25.1019,E2 -219.8007} C_DIS
LIN {X 27.7391,Y -36.7353,Z 63,A -59.8541,B 24.8719,C -2.6119,E1 25.0949,E2 -216.6309} C_DIS
LIN {X 25.4503,Y -38.3566,Z 63,A -63.4078,B 24.8727,C -2.604,E1 25.0867,E2 -213.0704} C_DIS
LIN {X 23.0559,Y -39.8419,Z 63,A -67.4982,B 24.8743,C -2.5875,E1 25.0769,E2 -208.9537} C_DIS
LIN {X 20.5441,Y -41.1932,Z 63,A -70.4408,B 24.8738,C -2.5922,E1 25.0696,E2 -206.0302} C_DIS
LIN {X 18.1742,Y -42.2928,Z 63,A -73.6532,B 24.8743,C -2.588,E1 25.0614,E2 -202.8158} C_DIS
LIN {X 15.9283,Y -43.1885,Z 63,A -76.6443,B 24.8746,C -2.5843,E1 25.0536,E2 -199.8224} C_DIS
LIN {X 13.5811,Y -43.9828,Z 63,A -80.6735,B 24.8765,C -2.565,E1 25.0428,E2 -195.7548} C_DIS
LIN {X 9.4366,Y -45.0545,Z 63,A -84.9705,B 24.8753,C -2.5769,E1 25.0312,E2 -191.4921} C_DIS
LIN {X 7.0252,Y -45.4926,Z 63,A -88.0403,B 24.8756,C -2.5743,E1 25.0227,E2 -188.4194} C_DIS
LIN {X 4.7331,Y -45.7879,Z 63,A -90.9745,B 24.8758,C -2.5717,E1 25.0146,E2 -185.4812} C_DIS
LIN {X 2.1883,Y -45.9803,Z 63,A -94.2025,B 24.8761,C -2.5695,E1 25.0056,E2 -182.2493} C_DIS
LIN {X 0.2175,Y -46.0213,Z 63,A -96.2949,B 24.8755,C -2.5747,E1 24.9998,E2 -180.1696} C_DIS
Enddeposition()
LIN {X 0.2175,Y -46.0213,Z 63,A -96.2949,B 24.8755,C -2.5747,E1 24.9998,E2 -180.1696} C_DIS
Startdeposition()
$VEL.CP = VEL_PRINT
LIN {X 0.3535,Y -45.0807,Z 63,A -94.6131,B 24.8716,C -2.615,E1 25.0047,E2 -181.947} C_DIS
LIN {X 3.4078,Y -44.9534,Z 63,A -91.0918,B 24.872,C -2.6108,E1 25.0145,E2 -185.4567} C_DIS
LIN {X 5.7996,Y -44.7074,Z 63,A -87.9812,B 24.8718,C -2.6135,E1 25.0232,E2 -188.5715} C_DIS
LIN {X 7.6913,Y -44.4218,Z 63,A -85.3895,B 24.8713,C -2.6179,E1 25.0303,E2 -191.171} C_DIS
LIN {X 11.0451,Y -43.7084,Z 63,A -81.1167,B 24.8711,C -2.6205,E1 25.0419,E2 -195.4442} C_DIS
LIN {X 13.3985,Y -43.0449,Z 63,A -77.6505,B 24.8701,C -2.6301,E1 25.0512,E2 -198.9269} C_DIS
LIN {X 16.5926,Y -41.9176,Z 63,A -73.8786,B 24.8705,C -2.6266,E1 25.0611,E2 -202.6826} C_DIS
LIN {X 18.7972,Y -40.977,Z 63,A -71.0997,B 24.8705,C -2.6266,E1 25.0682,E2 -205.4545} C_DIS
LIN {X 21.1519,Y -39.8112,Z 63,A -67.3046,B 24.8691,C -2.6399,E1 25.0776,E2 -209.2709} C_DIS
LIN {X 23.3027,Y -38.5918,Z 63,A -64.193,B 24.8686,C -2.645,E1 25.0851,E2 -212.385} C_DIS
LIN {X 25.4692,Y -37.1989,Z 63,A -61.1689,B 24.8684,C -2.6469,E1 25.0922,E2 -215.4036} C_DIS
LIN {X 27.0919,Y -36.0335,Z 63,A -58.7629,B 24.8682,C -2.6497,E1 25.0976,E2 -217.8078} C_DIS
LIN {X 28.9282,Y -34.5769,Z 63,A -55.9699,B 24.8679,C -2.6528,E1 25.1036,E2 -220.5975} C_DIS
LIN {X 31.0186,Y -32.7149,Z 63,A -51.4167,B 24.8652,C -2.6789,E1 25.1131,E2 -225.194} C_DIS
LIN {X 33.4813,Y -30.1896,Z 63,A -47.666,B 24.8655,C -2.6765,E1 25.1202,E2 -228.9227} C_DIS
LIN {X 35.087,Y -28.3072,Z 63,A -44.4889,B 24.8646,C -2.6852,E1 25.1259,E2 -232.1057} C_DIS
LIN {X 36.7914,Y -26.053,Z 63,A -41.076,B 24.864,C -2.6914,E1 25.1315,E2 -235.517} C_DIS
LIN {X 37.9442,Y -24.3438,Z 63,A -38.3318,B 24.863,C -2.7009,E1 25.1357,E2 -238.27} C_DIS
LIN {X 39.2391,Y -22.1978,Z 63,A -35.0911,B 24.862,C -2.7109,E1 25.1403,E2 -241.5177} C_DIS
LIN {X 40.4316,Y -19.942,Z 63,A -32.3598,B 24.862,C -2.7109,E1 25.1438,E2 -244.2342} C_DIS
LIN {X 41.3985,Y -17.849,Z 63,A -28.7237,B 24.8598,C -2.7326,E1 25.148,E2 -247.9021} C_DIS
LIN {X 42.3375,Y -15.4894,Z 63,A -25.6244,B 24.859,C -2.7399,E1 25.151,E2 -251.0015} C_DIS
LIN {X 43.2429,Y -12.7451,Z 63,A -22.5267,B 24.859,C -2.7404,E1 25.1536,E2 -254.0828} C_DIS
LIN {X 43.6193,Y -11.3917,Z 63,A -20.3347,B 24.8576,C -2.7536,E1 25.1552,E2 -256.2931} C_DIS
LIN {X 44.2887,Y -8.4206,Z 63,A -16.2839,B 24.856,C -2.769,E1 25.1575,E2 -260.3569} C_DIS
LIN {X 44.7217,Y -5.6887,Z 63,A -13.0293,B 24.8553,C -2.7751,E1 25.1588,E2 -263.6068} C_DIS
LIN {X 44.9458,Y -3.5026,Z 63,A -10.2121,B 24.8544,C -2.7844,E1 25.1595,E2 -266.4292} C_DIS
LIN {X 45.0721,Y -0.9487,Z 63,A -7.083,B 24.8535,C -2.7923,E1 25.1598,E2 -269.5585} C_DIS
LIN {X 45.0494,Y 1.713,Z 63,A -3.6734,B 24.8524,C -2.8034,E1 25.1596,E2 -272.9741} C_DIS
LIN {X 44.9287,Y 3.7165,Z 63,A -1.4192,B 24.8521,C -2.8058,E1 25.1591,E2 -275.2206} C_DIS
LIN {X 44.7637,Y 5.3485,Z 63,A 0.6772,B 24.8514,C -2.8125,E1 25.1585,E2 -277.3204} C_DIS
LIN {X 44.5273,Y 7.052,Z 63,A 2.9418,B 24.8505,C -2.8207,E1 25.1575,E2 -279.591} C_DIS
LIN {X 44.1824,Y 8.9618,Z 63,A 6.2142,B 24.8481,C -2.8432,E1 25.1557,E2 -282.8977} C_DIS
LIN {X 43.3217,Y 12.476,Z 63,A 10.1207,B 24.8481,C -2.844,E1 25.1529,E2 -286.7836} C_DIS
LIN {X 42.7538,Y 14.3007,Z 63,A 13.0877,B 24.8462,C -2.8611,E1 25.1503,E2 -289.7742} C_DIS
LIN {X 41.3106,Y 18.0504,Z 63,A 17.602,B 24.8458,C -2.8646,E1 25.1456,E2 -294.2718} C_DIS
LIN {X 40.1726,Y 20.4577,Z 63,A 20.8899,B 24.845,C -2.872,E1 25.1415,E2 -297.5598} C_DIS
LIN {X 39.2808,Y 22.123,Z 63,A 23.4964,B 24.8439,C -2.8821,E1 25.138,E2 -300.1765} C_DIS
LIN {X 37.8069,Y 24.5572,Z 63,A 27.1806,B 24.8428,C -2.8926,E1 25.1325,E2 -303.8668} C_DIS
LIN {X 36.2302,Y 26.8295,Z 63,A 30.1854,B 24.8428,C -2.8919,E1 25.1276,E2 -306.8556} C_DIS
LIN {X 34.6561,Y 28.833,Z 63,A 33.4319,B 24.842,C -2.8996,E1 25.122,E2 -310.1052} C_DIS
LIN {X 33.5271,Y 30.1385,Z 63,A 36.0306,B 24.8407,C -2.9116,E1 25.1171,E2 -312.7208} C_DIS
LIN {X 31.0754,Y 32.6615,Z 63,A 40.8633,B 24.839,C -2.9272,E1 25.1075,E2 -317.5701} C_DIS
LIN {X 28.1924,Y 35.1801,Z 63,A 44.8423,B 24.8397,C -2.9209,E1 25.099,E2 -321.5186} C_DIS
LIN {X 26.6558,Y 36.3573,Z 63,A 47.6406,B 24.8386,C -2.9309,E1 25.0928,E2 -324.3307} C_DIS
LIN {X 23.6211,Y 38.3977,Z 63,A 51.7837,B 24.8387,C -2.9296,E1 25.0831,E2 -328.457} C_DIS
LIN {X 22.5166,Y 39.0563,Z 63,A 53.5943,B 24.8381,C -2.9349,E1 25.0788,E2 -330.2745} C_DIS
LIN {X 21.033,Y 39.8748,Z 63,A 55.8551,B 24.8376,C -2.9395,E1 25.0732,E2 -332.5398} C_DIS
LIN {X 19.2498,Y 40.766,Z 63,A 58.3936,B 24.8373,C -2.9426,E1 25.0668,E2 -335.0789} C_DIS
LIN {X 17.2901,Y 41.6341,Z 63,A 61.4736,B 24.8363,C -2.9513,E1 25.0589,E2 -338.1724} C_DIS
LIN {X 15.0113,Y 42.5094,Z 63,A 65.0856,B 24.8351,C -2.9624,E1 25.0493,E2 -341.8033} C_DIS
LIN {X 11.4164,Y 43.613,Z 63,A 69.1862,B 24.836,C -2.9546,E1 25.0384,E2 -345.8785} C_DIS
LIN {X 8.8447,Y 44.2064,Z 63,A 72.2903,B 24.8362,C -2.9522,E1 25.0299,E2 -348.9728} C_DIS
LIN {X 6.6891,Y 44.5834,Z 63,A 75.2359,B 24.8358,C -2.9556,E1 25.0218,E2 -351.9238} C_DIS
LIN {X 3.8301,Y 44.9196,Z 63,A 78.8971,B 24.8358,C -2.9561,E1 25.0116,E2 -355.5837} C_DIS
LIN {X 1.3398,Y 45.0621,Z 63,A 82.0749,B 24.8358,C -2.9561,E1 25.0028,E2 -358.7604} C_DIS
LIN {X -0.5653,Y 45.0792,Z 63,A 84.8503,B 24.8352,C -2.9609,E1 24.995,E2 -361.5474} C_DIS
LIN {X -4.0681,Y 44.8981,Z 63,A 88.6131,B 24.8366,C -2.9487,E1 24.9846,E2 -365.2825} C_DIS
LIN {X -6.3846,Y 44.6276,Z 63,A 91.9317,B 24.8362,C -2.9522,E1 24.9754,E2 -368.6118} C_DIS
LIN {X -8.848,Y 44.2057,Z 63,A 94.769,B 24.837,C -2.9449,E1 24.9676,E2 -371.4345} C_DIS
LIN {X -11.7851,Y 43.5143,Z 63,A 99.7721,B 24.8356,C -2.9581,E1 24.954,E2 -376.4764} C_DIS
LIN {X -15.0217,Y 42.5058,Z 63,A 103.0728,B 24.8377,C -2.9386,E1 24.9453,E2 -379.7368} C_DIS
LIN {X -16.5718,Y 41.9251,Z 63,A 105.5973,B 24.8374,C -2.9418,E1 24.9387,E2 -382.2742} C_DIS
LIN {X -19.6656,Y 40.5669,Z 63,A 109.635,B 24.8385,C -2.9318,E1 24.9285,E2 -386.2981} C_DIS
LIN {X -21.9321,Y 39.3874,Z 63,A 113.0798,B 24.8388,C -2.9291,E1 24.92,E2 -389.7463} C_DIS
LIN {X -23.9542,Y 38.1914,Z 63,A 115.5226,B 24.8402,C -2.9165,E1 24.9143,E2 -392.1663} C_DIS
LIN {X -26.4118,Y 36.5359,Z 63,A 119.8193,B 24.8402,C -2.9162,E1 24.9044,E2 -396.477} C_DIS
LIN {X -28.4687,Y 34.9561,Z 63,A 122.6588,B 24.8416,C -2.9033,E1 24.8982,E2 -399.2961} C_DIS
LIN {X -30.3865,Y 33.3026,Z 63,A 126.5856,B 24.8414,C -2.9054,E1 24.8899,E2 -403.2436} C_DIS
LIN {X -32.154,Y 31.5994,Z 63,A 129.113,B 24.843,C -2.8904,E1 24.8849,E2 -405.7457} C_DIS
LIN {X -33.4143,Y 30.2636,Z 63,A 131.9768,B 24.8429,C -2.8916,E1 24.8795,E2 -408.6249} C_DIS
LIN {X -35.2632,Y 28.0877,Z 63,A 135.2026,B 24.8445,C -2.8772,E1 24.8738,E2 -411.8312} C_DIS
LIN {X -37.0192,Y 25.7287,Z 63,A 139.6906,B 24.8445,C -2.8768,E1 24.8665,E2 -416.3402} C_DIS
LIN {X -38.3419,Y 23.7134,Z 63,A 142.6403,B 24.8456,C -2.8669,E1 24.8621,E2 -419.2812} C_DIS
LIN {X -40.1113,Y 20.5783,Z 63,A 146.8945,B 24.8474,C -2.8498,E1 24.8565,E2 -423.517} C_DIS
LIN {X -41.8141,Y 16.8519,Z 63,A 153.0442,B 24.8478,C -2.8462,E1 24.8497,E2 -429.692} C_DIS
LIN {X -43.2036,Y 12.8777,Z 63,A 157.183,B 24.8512,C -2.8148,E1 24.8461,E2 -433.7795} C_DIS
LIN {X -43.5852,Y 11.5226,Z 63,A 159.2855,B 24.8513,C -2.8132,E1 24.8446,E2 -435.8903} C_DIS
LIN {X -44.2289,Y 8.731,Z 63,A 162.7047,B 24.8528,C -2.7991,E1 24.8425,E2 -439.296} C_DIS
LIN {X -44.6852,Y 5.9658,Z 63,A 166.8345,B 24.8533,C -2.795,E1 24.8408,E2 -443.4405} C_DIS
LIN {X -44.9613,Y 3.2894,Z 63,A 170.2396,B 24.8544,C -2.7841,E1 24.84,E2 -446.8399} C_DIS
LIN {X -45.0807,Y 0.3428,Z 63,A 173.8293,B 24.8558,C -2.7703,E1 24.8398,E2 -450.4184} C_DIS
LIN {X -45.0313,Y -2.1481,Z 63,A 176.5389,B 24.8575,C -2.7548,E1 24.84,E2 -453.1072} C_DIS
LIN {X -44.9099,Y -3.9364,Z 63,A 179.1484,B 24.8578,C -2.7518,E1 24.8406,E2 -455.7251} C_DIS
LIN {X -44.6731,Y -6.0572,Z 63,A -177.7592,B 24.8581,C -2.7482,E1 24.8417,E2 -458.8273} C_DIS
LIN {X -44.1747,Y -8.9993,Z 63,A -174.1578,B 24.8596,C -2.7342,E1 24.8435,E2 -462.4167} C_DIS
LIN {X -43.6379,Y -11.3194,Z 63,A -170.7462,B 24.86,C -2.73,E1 24.8458,E2 -465.8382} C_DIS
LIN {X -42.5022,Y -15.0318,Z 63,A -165.8171,B 24.8615,C -2.7156,E1 24.8501,E2 -470.7609} C_DIS
LIN {X -41.0481,Y -18.6402,Z 63,A -160.9353,B 24.863,C -2.7009,E1 24.8554,E2 -475.6346} C_DIS
LIN {X -39.4074,Y -21.8964,Z 63,A -156.4837,B 24.8645,C -2.6862,E1 24.8612,E2 -480.0747} C_DIS
LIN {X -38.1035,Y -24.0951,Z 63,A -153.3081,B 24.8654,C -2.6769,E1 24.8658,E2 -483.2443} C_DIS
LIN {X -35.9701,Y -27.1759,Z 63,A -148.6277,B 24.8667,C -2.6642,E1 24.8734,E2 -487.9175} C_DIS
LIN {X -34.3974,Y -29.1414,Z 63,A -144.7826,B 24.8666,C -2.6655,E1 24.8803,E2 -491.7834} C_DIS
LIN {X -32.6254,Y -31.1126,Z 63,A -141.881,B 24.8679,C -2.652,E1 24.8857,E2 -494.6655} C_DIS
LIN {X -30.8425,Y -32.8805,Z 63,A -138.4715,B 24.8683,C -2.6486,E1 24.8926,E2 -498.0809} C_DIS
LIN {X -28.851,Y -34.6411,Z 63,A -135.2154,B 24.8691,C -2.6406,E1 24.8995,E2 -501.3305} C_DIS
LIN {X -26.7065,Y -36.3202,Z 63,A -131.7343,B 24.8696,C -2.6349,E1 24.9073,E2 -504.8106} C_DIS
LIN {X -24.976,Y -37.5316,Z 63,A -129.2739,B 24.8704,C -2.6275,E1 24.9129,E2 -507.2617} C_DIS
LIN {X -22.8036,Y -38.8896,Z 63,A -125.928,B 24.8707,C -2.6241,E1 24.9209,E2 -510.6097} C_DIS
LIN {X -20.8187,Y -39.9876,Z 63,A -122.9122,B 24.8709,C -2.6223,E1 24.9283,E2 -513.6297} C_DIS
LIN {X -18.4979,Y -41.1122,Z 63,A -120.0474,B 24.8718,C -2.6126,E1 24.9355,E2 -516.4788} C_DIS
LIN {X -15.6535,Y -42.2777,Z 63,A -115.6848,B 24.8716,C -2.6156,E1 24.9469,E2 -520.8578} C_DIS
LIN {X -13.291,Y -43.0783,Z 63,A -112.5655,B 24.8719,C -2.6124,E1 24.9552,E2 -523.9754} C_DIS
LIN {X -10.877,Y -43.7506,Z 63,A -109.3359,B 24.8719,C -2.6113,E1 24.9639,E2 -527.207} C_DIS
LIN {X -7.1856,Y -44.5063,Z 63,A -104.5371,B 24.8721,C -2.6097,E1 24.9771,E2 -532.0071} C_DIS
LIN {X -4.7737,Y -44.8286,Z 63,A -101.5178,B 24.8723,C -2.6081,E1 24.9854,E2 -535.0247} C_DIS
LIN {X -2.2965,Y -45.0239,Z 63,A -98.2895,B 24.8722,C -2.6093,E1 24.9944,E2 -538.2569} C_DIS
LIN {X 0.2242,Y -45.0797,Z 63,A -96.5395,B 24.8743,C -2.5871,E1 24.9992,E2 -539.9544} C_DIS
Enddeposition()
LIN {X 0.2242,Y -45.0797,Z 63,A -96.5395,B 24.8743,C -2.5871,E1 24.9992,E2 -539.9544} C_DIS
Startdeposition()
$VEL.CP = VEL_PRINT
LIN {X -0.8281,Y -44.1244,Z 63,A -98.2699,B 24.8733,C -2.598,E1 24.9944,E2 -538.2499} C_DIS
LIN {X -3.1358,Y -44.0209,Z 63,A -101.0628,B 24.873,C -2.601,E1 24.9866,E2 -535.463} C_DIS
LIN {X -5.5129,Y -43.7867,Z 63,A -104.1136,B 24.8729,C -2.6021,E1 24.9782,E2 -532.413} C_DIS
LIN {X -8.2948,Y -43.3456,Z 63,A -107.8019,B 24.8729,C -2.6028,E1 24.968,E2 -528.7227} C_DIS
LIN {X -11.1378,Y -42.7039,Z 63,A -111.5513,B 24.8726,C -2.6052,E1 24.9579,E2 -524.9739} C_DIS
LIN {X -13.5116,Y -42.013,Z 63,A -114.7979,B 24.8724,C -2.6069,E1 24.9492,E2 -521.7259} C_DIS
LIN {X -16.2242,Y -41.0418,Z 63,A -118.8339,B 24.8724,C -2.6062,E1 24.9386,E2 -517.6796} C_DIS
LIN {X -19.7459,Y -39.4679,Z 63,A -123.8003,B 24.8719,C -2.6124,E1 24.9261,E2 -512.7157} C_DIS
LIN {X -21.814,Y -38.3644,Z 63,A -126.3654,B 24.8708,C -2.6229,E1 24.9198,E2 -510.1682} C_DIS
LIN {X -24.2997,Y -36.8398,Z 63,A -130.8092,B 24.8711,C -2.6197,E1 24.9093,E2 -505.7027} C_DIS
LIN {X -27.1515,Y -34.7925,Z 63,A -134.6008,B 24.8694,C -2.6375,E1 24.9008,E2 -501.94} C_DIS
LIN {X -28.5691,Y -33.6371,Z 63,A -137.43,B 24.8695,C -2.6359,E1 24.8947,E2 -499.0963} C_DIS
LIN {X -30.2008,Y -32.1801,Z 63,A -140.7454,B 24.8695,C -2.6354,E1 24.8879,E2 -495.7662} C_DIS
LIN {X -32.391,Y -29.975,Z 63,A -144.5436,B 24.8684,C -2.647,E1 24.8806,E2 -491.9791} C_DIS
LIN {X -34.6995,Y -27.2692,Z 63,A -149.289,B 24.8675,C -2.6559,E1 24.8722,E2 -487.2331} C_DIS
LIN {X -36.7908,Y -24.3741,Z 63,A -153.396,B 24.8658,C -2.6738,E1 24.8657,E2 -483.1486} C_DIS
LIN {X -37.9745,Y -22.4852,Z 63,A -156.5922,B 24.8654,C -2.6775,E1 24.861,E2 -479.9449} C_DIS
LIN {X -39.3983,Y -19.8843,Z 63,A -160.9323,B 24.8649,C -2.682,E1 24.8554,E2 -475.5924} C_DIS
LIN {X -41.0438,Y -16.2191,Z 63,A -165.76,B 24.863,C -2.7012,E1 24.8501,E2 -470.7838} C_DIS
LIN {X -41.7549,Y -14.2903,Z 63,A -168.4883,B 24.8623,C -2.7082,E1 24.8476,E2 -468.0568} C_DIS
LIN {X -42.5209,Y -11.8168,Z 63,A -171.8038,B 24.8612,C -2.7186,E1 24.845,E2 -464.747} C_DIS
LIN {X -43.1084,Y -9.4506,Z 63,A -174.9069,B 24.8601,C -2.7288,E1 24.8431,E2 -461.6503} C_DIS
LIN {X -43.6793,Y -6.3055,Z 63,A -179.1634,B 24.859,C -2.7403,E1 24.8411,E2 -457.3959} C_DIS
LIN {X -43.988,Y -3.5553,Z 63,A 176.9379,B 24.8582,C -2.7479,E1 24.8401,E2 -453.4921} C_DIS
LIN {X -44.1302,Y -0.4557,Z 63,A 173.1902,B 24.8565,C -2.7637,E1 24.8398,E2 -449.7596} C_DIS
LIN {X -44.0488,Y 2.7091,Z 63,A 168.9768,B 24.8553,C -2.7755,E1 24.8403,E2 -445.5489} C_DIS
LIN {X -43.821,Y 5.232,Z 63,A 165.7695,B 24.8541,C -2.7867,E1 24.8412,E2 -442.3493} C_DIS
LIN {X -43.4233,Y 7.8781,Z 63,A 162.236,B 24.8531,C -2.7969,E1 24.8428,E2 -438.8191} C_DIS
LIN {X -42.8862,Y 10.4126,Z 63,A 158.9441,B 24.8519,C -2.8081,E1 24.8448,E2 -435.5348} C_DIS
LIN {X -42.3378,Y 12.4567,Z 63,A 156.2526,B 24.8509,C -2.8172,E1 24.8469,E2 -432.8494} C_DIS
LIN {X -41.6607,Y 14.5615,Z 63,A 152.7003,B 24.8509,C -2.818,E1 24.8501,E2 -429.2789} C_DIS
LIN {X -40.0955,Y 18.4401,Z 63,A 147.8369,B 24.8484,C -2.8407,E1 24.8553,E2 -424.4428} C_DIS
LIN {X -39.2623,Y 20.1525,Z 63,A 145.6576,B 24.8473,C -2.8513,E1 24.858,E2 -422.2771} C_DIS
LIN {X -38.3122,Y 21.905,Z 63,A 142.6228,B 24.847,C -2.8534,E1 24.8622,E2 -419.2313} C_DIS
LIN {X -37.0306,Y 24.0083,Z 63,A 139.0909,B 24.8465,C -2.8582,E1 24.8675,E2 -415.6931} C_DIS
LIN {X -34.8328,Y 27.0991,Z 63,A 134.6762,B 24.8444,C -2.8773,E1 24.8747,E2 -411.3026} C_DIS
LIN {X -32.9561,Y 29.3522,Z 63,A 130.0308,B 24.8445,C -2.8767,E1 24.8832,E2 -406.6348} C_DIS
LIN {X -29.5966,Y 32.7373,Z 63,A 123.6478,B 24.8432,C -2.8887,E1 24.8961,E2 -400.2541} C_DIS
LIN {X -27.0428,Y 34.8762,Z 63,A 119.414,B 24.8421,C -2.8989,E1 24.9054,E2 -396.029} C_DIS
LIN {X -23.5302,Y 37.3364,Z 63,A 114.3863,B 24.8402,C -2.9163,E1 24.917,E2 -391.0262} C_DIS
LIN {X -20.8984,Y 38.8706,Z 63,A 110.5357,B 24.8393,C -2.9244,E1 24.9263,E2 -387.1837} C_DIS
LIN {X -18.998,Y 39.8339,Z 63,A 107.0615,B 24.8398,C -2.9195,E1 24.9351,E2 -383.6887} C_DIS
LIN {X -14.5957,Y 41.6487,Z 63,A 102.3407,B 24.8368,C -2.9472,E1 24.9472,E2 -379.0237} C_DIS
LIN {X -12.499,Y 42.3252,Z 63,A 98.5069,B 24.8379,C -2.9372,E1 24.9575,E2 -375.1593} C_DIS
LIN {X -10.1037,Y 42.9592,Z 63,A 95.3894,B 24.8374,C -2.9416,E1 24.9659,E2 -372.0479} C_DIS
LIN {X -8.3002,Y 43.3446,Z 63,A 92.522,B 24.8379,C -2.9369,E1 24.9738,E2 -369.1663} C_DIS
LIN {X -4.5297,Y 43.8991,Z 63,A 88.4091,B 24.8363,C -2.9516,E1 24.9851,E2 -365.0852} C_DIS
LIN {X -2.9108,Y 44.036,Z 63,A 86.0446,B 24.8366,C -2.9489,E1 24.9917,E2 -362.7133} C_DIS
LIN {X -0.3612,Y 44.1308,Z 63,A 83.1985,B 24.8357,C -2.9565,E1 24.9996,E2 -359.885} C_DIS
LIN {X 1.2312,Y 44.1151,Z 63,A 80.5815,B 24.8366,C -2.9488,E1 25.007,E2 -357.25} C_DIS
LIN {X 3.8322,Y 43.9659,Z 63,A 77.5129,B 24.8361,C -2.9533,E1 25.0155,E2 -354.1936} C_DIS
LIN {X 5.589,Y 43.7769,Z 63,A 75.1496,B 24.8362,C -2.9519,E1 25.022,E2 -351.8286} C_DIS
LIN {X 8.2198,Y 43.3601,Z 63,A 71.7104,B 24.8363,C -2.9511,E1 25.0315,E2 -348.391} C_DIS
LIN {X 10.2891,Y 42.9163,Z 63,A 68.6611,B 24.837,C -2.9451,E1 25.0398,E2 -345.3316} C_DIS
LIN {X 13.7898,Y 41.9227,Z 63,A 64.1208,B 24.837,C -2.9446,E1 25.052,E2 -340.7981} C_DIS
LIN {X 15.3609,Y 41.3732,Z 63,A 61.4468,B 24.8382,C -2.9346,E1 25.059,E2 -338.1061} C_DIS
LIN {X 18.5273,Y 40.0549,Z 63,A 57.2962,B 24.8382,C -2.9346,E1 25.0696,E2 -333.9654} C_DIS
LIN {X 21.2794,Y 38.6633,Z 63,A 53.5038,B 24.8384,C -2.9329,E1 25.079,E2 -330.1796} C_DIS
LIN {X 23.4928,Y 37.3598,Z 63,A 49.8404,B 24.8395,C -2.9227,E1 25.0877,E2 -326.5034} C_DIS
LIN {X 25.752,Y 35.84,Z 63,A 46.4048,B 24.8399,C -2.9185,E1 25.0956,E2 -323.0699} C_DIS
LIN {X 27.6062,Y 34.4325,Z 63,A 43.6038,B 24.8401,C -2.9168,E1 25.1017,E2 -320.2751} C_DIS
LIN {X 29.4362,Y 32.8809,Z 63,A 40.4336,B 24.8409,C -2.9099,E1 25.1084,E2 -317.1011} C_DIS
LIN {X 31.2793,Y 31.1328,Z 63,A 37.2377,B 24.8414,C -2.9049,E1 25.1148,E2 -313.9067} C_DIS
LIN {X 32.8614,Y 29.458,Z 63,A 34.2714,B 24.8421,C -2.8988,E1 25.1204,E2 -310.939} C_DIS
LIN {X 35.1041,Y 26.7471,Z 63,A 30.1188,B 24.8425,C -2.8954,E1 25.1277,E2 -306.7976} C_DIS
LIN {X 37.1557,Y 23.8138,Z 63,A 25.3373,B 24.844,C -2.8816,E1 25.1353,E2 -302.007} C_DIS
LIN {X 38.0195,Y 22.4091,Z 63,A 22.6809,B 24.8456,C -2.8671,E1 25.1392,E2 -299.3298} C_DIS
LIN {X 39.0505,Y 20.5598,Z 63,A 19.7214,B 24.8467,C -2.8561,E1 25.1431,E2 -296.3598} C_DIS
LIN {X 40.2626,Y 18.0713,Z 63,A 16.8384,B 24.8465,C -2.8587,E1 25.1464,E2 -293.4985} C_DIS
LIN {X 41.0004,Y 16.3296,Z 63,A 13.0826,B 24.8497,C -2.8289,E1 25.1504,E2 -289.6929} C_DIS
LIN {X 42.4024,Y 12.2362,Z 63,A 8.5608,B 24.8494,C -2.8317,E1 25.1542,E2 -285.2036} C_DIS
LIN {X 43.1649,Y 9.1878,Z 63,A 4.9139,B 24.8498,C -2.8272,E1 25.1565,E2 -281.5671} C_DIS
LIN {X 43.4253,Y 7.8674,Z 63,A 2.7941,B 24.8511,C -2.8152,E1 25.1576,E2 -279.4313} C_DIS
LIN {X 43.81,Y 5.326,Z 63,A -0.504,B 24.8521,C -2.8056,E1 25.1589,E2 -276.1299} C_DIS
LIN {X 44.0721,Y 2.3055,Z 63,A -4.8443,B 24.8542,C -2.7862,E1 25.1597,E2 -271.7693} C_DIS
LIN {X 44.1199,Y -1.0716,Z 63,A -8.7543,B 24.8547,C -2.7809,E1 25.1597,E2 -267.8702} C_DIS
LIN {X 43.9923,Y -3.5101,Z 63,A -11.7965,B 24.8555,C -2.7733,E1 25.1591,E2 -264.8279} C_DIS
LIN {X 43.7331,Y -5.9178,Z 63,A -14.9037,B 24.8565,C -2.7641,E1 25.1581,E2 -261.7173} C_DIS
LIN {X 43.3697,Y -8.1699,Z 63,A -18.0359,B 24.8578,C -2.7517,E1 25.1566,E2 -258.5743} C_DIS
LIN {X 42.926,Y -10.2494,Z 63,A -20.5386,B 24.8582,C -2.7478,E1 25.155,E2 -256.0767} C_DIS
LIN {X 42.4608,Y -12.0302,Z 63,A -22.915,B 24.8589,C -2.7406,E1 25.1533,E2 -253.6972} C_DIS
LIN {X 41.9033,Y -13.8495,Z 63,A -25.4314,B 24.8598,C -2.7322,E1 25.1512,E2 -251.1752} C_DIS
LIN {X 41.1321,Y -15.9945,Z 63,A -28.4013,B 24.8607,C -2.7231,E1 25.1483,E2 -248.2002} C_DIS
LIN {X 40.3086,Y -17.9678,Z 63,A -31.4023,B 24.862,C -2.7109,E1 25.1449,E2 -245.1867} C_DIS
LIN {X 39.161,Y -20.35,Z 63,A -35.0853,B 24.8635,C -2.6965,E1 25.1403,E2 -241.4891} C_DIS
LIN {X 37.5714,Y -23.1537,Z 63,A -38.5886,B 24.8635,C -2.6967,E1 25.1353,E2 -238.0046} C_DIS
LIN {X 36.7305,Y -24.4651,Z 63,A -40.9321,B 24.8646,C -2.6855,E1 25.1317,E2 -235.6461} C_DIS
LIN {X 35.0171,Y -26.86,Z 63,A -44.5012,B 24.8651,C -2.6798,E1 25.1258,E2 -232.0807} C_DIS
LIN {X 33.6226,Y -28.5861,Z 63,A -47.5262,B 24.8661,C -2.6699,E1 25.1204,E2 -229.0462} C_DIS
LIN {X 31.967,Y -30.4271,Z 63,A -51.3241,B 24.8679,C -2.6519,E1 25.1131,E2 -225.2224} C_DIS
LIN {X 28.7459,Y -33.4862,Z 63,A -56.4234,B 24.8681,C -2.6502,E1 25.1026,E2 -220.1397} C_DIS
LIN {X 26.4447,Y -35.3317,Z 63,A -60.4043,B 24.8692,C -2.6396,E1 25.0938,E2 -216.1483} C_DIS
LIN {X 24.6179,Y -36.6283,Z 63,A -63.6082,B 24.8702,C -2.629,E1 25.0864,E2 -212.93} C_DIS
LIN {X 21.976,Y -38.2714,Z 63,A -67.7636,B 24.8711,C -2.6198,E1 25.0764,E2 -208.7656} C_DIS
LIN {X 17.7134,Y -40.4214,Z 63,A -72.937,B 24.8704,C -2.6269,E1 25.0635,E2 -203.6228} C_DIS
LIN {X 14.7411,Y -41.5976,Z 63,A -78.1212,B 24.8726,C -2.6047,E1 25.0498,E2 -198.3969} C_DIS
LIN {X 11.9981,Y -42.4699,Z 63,A -80.8934,B 24.8715,C -2.6159,E1 25.0425,E2 -195.6563} C_DIS
LIN {X 9.8661,Y -43.0151,Z 63,A -83.8713,B 24.872,C -2.6112,E1 25.0344,E2 -192.6716} C_DIS
LIN {X 8.028,Y -43.3958,Z 63,A -86.3996,B 24.8723,C -2.6078,E1 25.0275,E2 -190.138} C_DIS
LIN {X 5.8417,Y -43.7441,Z 63,A -89.4149,B 24.8727,C -2.6036,E1 25.0191,E2 -187.1156} C_DIS
LIN {X 3.3449,Y -44.0055,Z 63,A -92.829,B 24.8731,C -2.5996,E1 25.0096,E2 -183.6939} C_DIS
LIN {X 0.9376,Y -44.1224,Z 63,A -96.0884,B 24.8734,C -2.5966,E1 25.0005,E2 -180.4281} C_DIS
LIN {X 0.9376,Y -44.1224,Z 63,A -96.0884,B 24.8734,C -2.5966,E1 25.0005,E2 -180.4281} C_DIS
Enddeposition()
LIN {X 0.2213,Y -43.1762,Z 63,A -96.1134,B 24.8705,C -2.6267,E1 25.0006,E2 -180.4747} C_DIS
Startdeposition()
$VEL.CP = VEL_PRINT
LIN {X 1.591,Y -43.1537,Z 63,A -93.2474,B 24.8688,C -2.6431,E1 25.0087,E2 -183.3789} C_DIS
LIN {X 4.7722,Y -42.9185,Z 63,A -89.0665,B 24.8687,C -2.6444,E1 25.0204,E2 -187.5606} C_DIS
LIN {X 7.5773,Y -42.5124,Z 63,A -85.4028,B 24.8686,C -2.6456,E1 25.0305,E2 -191.2235} C_DIS
LIN {X 9.8554,Y -42.0424,Z 63,A -82.0481,B 24.8679,C -2.6527,E1 25.0396,E2 -194.5905} C_DIS
LIN {X 11.8113,Y -41.5356,Z 63,A -79.5823,B 24.8679,C -2.652,E1 25.0463,E2 -197.0509} C_DIS
LIN {X 13.9296,Y -40.8735,Z 63,A -76.5402,B 24.8674,C -2.6571,E1 25.0543,E2 -200.0993} C_DIS
LIN {X 16.8434,Y -39.762,Z 63,A -72.8186,B 24.8675,C -2.656,E1 25.064,E2 -203.8099} C_DIS
LIN {X 18.3966,Y -39.0676,Z 63,A -70.5522,B 24.8672,C -2.6596,E1 25.0697,E2 -206.079} C_DIS
LIN {X 20.3212,Y -38.1021,Z 63,A -67.4085,B 24.8662,C -2.669,E1 25.0776,E2 -209.2364} C_DIS
LIN {X 22.8534,Y -36.6392,Z 63,A -63.0155,B 24.8646,C -2.6847,E1 25.0881,E2 -213.6529} C_DIS
LIN {X 25.0191,Y -35.1961,Z 63,A -60.3199,B 24.8653,C -2.6787,E1 25.0942,E2 -216.3249} C_DIS
LIN {X 26.8801,Y -33.7963,Z 63,A -57.0328,B 24.8643,C -2.6885,E1 25.1015,E2 -219.6233} C_DIS
LIN {X 28.5804,Y -32.3717,Z 63,A -53.9227,B 24.8633,C -2.6979,E1 25.1081,E2 -222.7435} C_DIS
LIN {X 30.826,Y -30.2403,Z 63,A -50.2649,B 24.8631,C -2.6998,E1 25.1154,E2 -226.3904} C_DIS
LIN {X 32.4165,Y -28.529,Z 63,A -46.9249,B 24.8619,C -2.7117,E1 25.1217,E2 -229.7437} C_DIS
LIN {X 33.9603,Y -26.6726,Z 63,A -43.3462,B 24.8604,C -2.7266,E1 25.128,E2 -233.341} C_DIS
LIN {X 36.1125,Y -23.6772,Z 63,A -39.1621,B 24.8604,C -2.7272,E1 25.1346,E2 -237.5061} C_DIS
LIN {X 37.4627,Y -21.477,Z 63,A -35.1625,B 24.8583,C -2.7471,E1 25.1403,E2 -241.5322} C_DIS
LIN {X 38.7657,Y -19.0253,Z 63,A -32.0037,B 24.8581,C -2.7483,E1 25.1443,E2 -244.6771} C_DIS
LIN {X 39.6383,Y -17.1329,Z 63,A -29.2294,B 24.8573,C -2.7567,E1 25.1475,E2 -247.4561} C_DIS
LIN {X 40.4185,Y -15.2007,Z 63,A -26.4146,B 24.8563,C -2.7659,E1 25.1503,E2 -250.2771} C_DIS
LIN {X 41.1385,Y -13.1289,Z 63,A -23.4453,B 24.8553,C -2.7758,E1 25.153,E2 -253.2531} C_DIS
LIN {X 41.805,Y -10.8193,Z 63,A -20.3976,B 24.8545,C -2.7831,E1 25.1552,E2 -256.3006} C_DIS
LIN {X 42.301,Y -8.6796,Z 63,A -17.7464,B 24.8541,C -2.7874,E1 25.1568,E2 -258.9465} C_DIS
LIN {X 42.5866,Y -7.1482,Z 63,A -15.1273,B 24.8523,C -2.8039,E1 25.158,E2 -261.5892} C_DIS
LIN {X 43.0259,Y -3.6796,Z 63,A -10.7471,B 24.8513,C -2.8137,E1 25.1594,E2 -265.9668} C_DIS
LIN {X 43.166,Y -1.1947,Z 63,A -7.1051,B 24.8495,C -2.8303,E1 25.1598,E2 -269.6263} C_DIS
LIN {X 43.1013,Y 2.6472,Z 63,A -2.0059,B 24.8478,C -2.8462,E1 25.1592,E2 -274.733} C_DIS
LIN {X 42.8438,Y 5.3984,Z 63,A 1.2666,B 24.8474,C -2.8504,E1 25.1582,E2 -277.996} C_DIS
LIN {X 42.4841,Y 7.7344,Z 63,A 4.0931,B 24.8469,C -2.8545,E1 25.1569,E2 -280.8155} C_DIS
LIN {X 42.1437,Y 9.4146,Z 63,A 6.8577,B 24.8452,C -2.8701,E1 25.1553,E2 -283.6011} C_DIS
LIN {X 41.4127,Y 12.2352,Z 63,A 10.0468,B 24.8452,C -2.8695,E1 25.1529,E2 -286.7705} C_DIS
LIN {X 40.6766,Y 14.4974,Z 63,A 13.9355,B 24.8429,C -2.8917,E1 25.1494,E2 -290.6897} C_DIS
LIN {X 39.6652,Y 17.0701,Z 63,A 17.4343,B 24.8421,C -2.899,E1 25.1457,E2 -294.1867} C_DIS
LIN {X 38.343,Y 19.8635,Z 63,A 21.0634,B 24.8418,C -2.9019,E1 25.1412,E2 -297.8031} C_DIS
LIN {X 37.3795,Y 21.6217,Z 63,A 23.9588,B 24.8405,C -2.913,E1 25.1372,E2 -300.7097} C_DIS
LIN {X 36.504,Y 23.0698,Z 63,A 26.9795,B 24.8384,C -2.9323,E1 25.1327,E2 -303.7608} C_DIS
LIN {X 34.4324,Y 26.0605,Z 63,A 31.1817,B 24.8384,C -2.933,E1 25.1258,E2 -307.9446} C_DIS
LIN {X 32.5388,Y 28.389,Z 63,A 34.498,B 24.8386,C -2.9308,E1 25.1199,E2 -311.2402} C_DIS
LIN {X 31.4648,Y 29.5748,Z 63,A 37.0438,B 24.8373,C -2.9425,E1 25.115,E2 -313.8028} C_DIS
LIN {X 29.735,Y 31.3143,Z 63,A 40.0988,B 24.8369,C -2.9458,E1 25.1089,E2 -316.8527} C_DIS
LIN {X 27.7195,Y 33.1107,Z 63,A 43.6131,B 24.8363,C -2.9515,E1 25.1016,E2 -320.3667} C_DIS
LIN {X 24.9538,Y 35.2426,Z 63,A 48.314,B 24.8353,C -2.9606,E1 25.0911,E2 -325.0722} C_DIS
LIN {X 22.8373,Y 36.6493,Z 63,A 52.038,B 24.8341,C -2.9715,E1 25.0823,E2 -328.81} C_DIS
LIN {X 21.1214,Y 37.6644,Z 63,A 54.3398,B 24.8343,C -2.9696,E1 25.0767,E2 -331.1004} C_DIS
LIN {X 18.9845,Y 38.7854,Z 63,A 57.7305,B 24.8335,C -2.9766,E1 25.0683,E2 -334.4984} C_DIS
LIN {X 16.7858,Y 39.7863,Z 63,A 60.8891,B 24.8332,C -2.9793,E1 25.0602,E2 -337.6558} C_DIS
LIN {X 14.6233,Y 40.6313,Z 63,A 64.0924,B 24.8326,C -2.9841,E1 25.0518,E2 -340.8635} C_DIS
LIN {X 12.1071,Y 41.4507,Z 63,A 67.7365,B 24.8321,C -2.9887,E1 25.0421,E2 -344.5121} C_DIS
LIN {X 9.2437,Y 42.1814,Z 63,A 71.0541,B 24.8329,C -2.9816,E1 25.0331,E2 -347.8081} C_DIS
LIN {X 6.341,Y 42.715,Z 63,A 75.4382,B 24.832,C -2.9899,E1 25.021,E2 -352.2074} C_DIS
LIN {X 4.0768,Y 42.9896,Z 63,A 78.17,B 24.8324,C -2.986,E1 25.0134,E2 -354.928} C_DIS
LIN {X 1.5263,Y 43.1558,Z 63,A 81.7549,B 24.8321,C -2.9887,E1 25.0034,E2 -358.5182} C_DIS
LIN {X -0.157,Y 43.1822,Z 63,A 84.1774,B 24.8319,C -2.991,E1 24.9967,E2 -360.9461} C_DIS
LIN {X -3.0473,Y 43.0749,Z 63,A 87.8127,B 24.8323,C -2.9867,E1 24.9865,E2 -364.5721} C_DIS
LIN {X -5.2623,Y 42.8611,Z 63,A 90.6266,B 24.8327,C -2.9831,E1 24.9788,E2 -367.3793} C_DIS
LIN {X -7.9046,Y 42.4529,Z 63,A 94.2511,B 24.8329,C -2.9817,E1 24.9688,E2 -371.0039} C_DIS
LIN {X -9.5597,Y 42.1106,Z 63,A 97.0293,B 24.8323,C -2.9872,E1 24.9612,E2 -373.7987} C_DIS
LIN {X -13.4117,Y 41.0469,Z 63,A 101.5147,B 24.8342,C -2.9704,E1 24.9492,E2 -378.2514} C_DIS
LIN {X -14.8018,Y 40.5662,Z 63,A 104.2295,B 24.8333,C -2.9782,E1 24.942,E2 -380.9903} C_DIS
LIN {X -18.329,Y 39.0995,Z 63,A 108.4805,B 24.8353,C -2.9601,E1 24.9312,E2 -385.2082} C_DIS
LIN {X -19.5124,Y 38.5227,Z 63,A 110.4539,B 24.8353,C -2.9603,E1 24.9263,E2 -387.1872} C_DIS
LIN {X -21.1409,Y 37.6532,Z 63,A 112.9903,B 24.8356,C -2.9573,E1 24.9201,E2 -389.7238} C_DIS
LIN {X -22.88,Y 36.6226,Z 63,A 116.136,B 24.8356,C -2.9585,E1 24.9126,E2 -392.882} C_DIS
LIN {X -25.838,Y 34.5994,Z 63,A 120.2242,B 24.8375,C -2.9406,E1 24.9033,E2 -396.9417} C_DIS
LIN {X -27.3018,Y 33.4566,Z 63,A 122.7289,B 24.838,C -2.936,E1 24.8978,E2 -399.4446} C_DIS
LIN {X -29.435,Y 31.5953,Z 63,A 127.1945,B 24.838,C -2.9364,E1 24.8885,E2 -403.929} C_DIS
LIN {X -31.9116,Y 29.0921,Z 63,A 132.0659,B 24.8389,C -2.9276,E1 24.8792,E2 -408.8006} C_DIS
LIN {X -34.0572,Y 26.5495,Z 63,A 136.4268,B 24.8403,C -2.9156,E1 24.8716,E2 -413.1531} C_DIS
LIN {X -35.7411,Y 24.234,Z 63,A 139.7396,B 24.842,C -2.8996,E1 24.8663,E2 -416.4439} C_DIS
LIN {X -36.9328,Y 22.376,Z 63,A 142.4372,B 24.8432,C -2.8887,E1 24.8623,E2 -419.1294} C_DIS
LIN {X -37.7352,Y 20.9942,Z 63,A 144.7549,B 24.8436,C -2.8851,E1 24.8591,E2 -421.4505} C_DIS
LIN {X -38.708,Y 19.1418,Z 63,A 147.3543,B 24.8447,C -2.875,E1 24.8558,E2 -424.0396} C_DIS
LIN {X -39.3664,Y 17.7481,Z 63,A 150.0085,B 24.8446,C -2.8762,E1 24.8527,E2 -426.7112} C_DIS
LIN {X -40.5882,Y 14.7412,Z 63,A 153.9167,B 24.8465,C -2.8586,E1 24.8488,E2 -430.5993} C_DIS
LIN {X -41.2637,Y 12.7289,Z 63,A 156.8046,B 24.8473,C -2.8509,E1 24.8463,E2 -433.4852} C_DIS
LIN {X -41.7501,Y 11.0308,Z 63,A 158.9183,B 24.8484,C -2.841,E1 24.8448,E2 -435.5875} C_DIS
LIN {X -42.173,Y 9.2821,Z 63,A 161.6517,B 24.8487,C -2.8376,E1 24.8431,E2 -438.3288} C_DIS
LIN {X -42.6145,Y 6.981,Z 63,A 165.0123,B 24.8495,C -2.8308,E1 24.8414,E2 -441.6932} C_DIS
LIN {X -42.9989,Y 3.9761,Z 63,A 168.5181,B 24.8514,C -2.8123,E1 24.8403,E2 -445.1756} C_DIS
LIN {X -43.1161,Y 2.3858,Z 63,A 171.7769,B 24.8507,C -2.819,E1 24.8398,E2 -448.47} C_DIS
LIN {X -43.1754,Y -0.7718,Z 63,A 175.9194,B 24.8522,C -2.8053,E1 24.8399,E2 -452.6046} C_DIS
LIN {X -42.9111,Y -4.8359,Z 63,A -178.9763,B 24.8543,C -2.785,E1 24.8412,E2 -457.6909} C_DIS
LIN {X -42.2417,Y -8.967,Z 63,A -174.0298,B 24.8568,C -2.7609,E1 24.8436,E2 -462.6093} C_DIS
LIN {X -41.8513,Y -10.6366,Z 63,A -171.2928,B 24.857,C -2.7596,E1 24.8455,E2 -465.3591} C_DIS
LIN {X -41.0019,Y -13.5493,Z 63,A -167.4219,B 24.8584,C -2.7459,E1 24.8486,E2 -469.2196} C_DIS
LIN {X -40.1765,Y -15.8291,Z 63,A -163.9736,B 24.859,C -2.7395,E1 24.8521,E2 -472.6719} C_DIS
LIN {X -38.7181,Y -19.1213,Z 63,A -159.0876,B 24.8603,C -2.7277,E1 24.8578,E2 -477.5562} C_DIS
LIN {X -37.5356,Y -21.3486,Z 63,A -155.8656,B 24.8613,C -2.7173,E1 24.8622,E2 -480.7705} C_DIS
LIN {X -36.106,Y -23.6871,Z 63,A -151.6745,B 24.8616,C -2.715,E1 24.8685,E2 -484.9773} C_DIS
LIN {X -34.0197,Y -26.5974,Z 63,A -148.0545,B 24.8642,C -2.6896,E1 24.8745,E2 -488.5539} C_DIS
LIN {X -32.7088,Y -28.1932,Z 63,A -144.6358,B 24.8639,C -2.6919,E1 24.8807,E2 -491.9939} C_DIS
LIN {X -31.2158,Y -29.8381,Z 63,A -142.0956,B 24.8651,C -2.6804,E1 24.8855,E2 -494.5178} C_DIS
LIN {X -29.9753,Y -31.0836,Z 63,A -139.6174,B 24.8654,C -2.6775,E1 24.8904,E2 -496.9994} C_DIS
LIN {X -28.545,Y -32.4017,Z 63,A -136.6887,B 24.8654,C -2.6771,E1 24.8965,E2 -499.9388} C_DIS
LIN {X -26.4861,Y -34.1061,Z 63,A -132.733,B 24.8655,C -2.6762,E1 24.9052,E2 -503.9069} C_DIS
LIN {X -24.1841,Y -35.7749,Z 63,A -129.9311,B 24.8674,C -2.6572,E1 24.9115,E2 -506.6731} C_DIS
LIN {X -22.8704,Y -36.6286,Z 63,A -127.7379,B 24.8676,C -2.6556,E1 24.9167,E2 -508.8696} C_DIS
LIN {X -21.2871,Y -37.5714,Z 63,A -125.1792,B 24.8678,C -2.6538,E1 24.9229,E2 -511.4315} C_DIS
LIN {X -19.1248,Y -38.7163,Z 63,A -121.4642,B 24.8675,C -2.6562,E1 24.9322,E2 -515.1623} C_DIS
LIN {X -17.1071,Y -39.6495,Z 63,A -118.8951,B 24.8684,C -2.6478,E1 24.9387,E2 -517.7176} C_DIS
LIN {X -13.7687,Y -40.9284,Z 63,A -114.0757,B 24.8687,C -2.6447,E1 24.9513,E2 -522.5394} C_DIS
LIN {X -11.5169,Y -41.619,Z 63,A -110.267,B 24.8679,C -2.6525,E1 24.9616,E2 -526.3728} C_DIS
LIN {X -8.4178,Y -42.354,Z 63,A -106.5109,B 24.8688,C -2.6438,E1 24.9718,E2 -530.1128} C_DIS
LIN {X -5.2397,Y -42.8638,Z 63,A -102.4048,B 24.8691,C -2.6404,E1 24.9832,E2 -534.2142} C_DIS
LIN {X -2.7549,Y -43.0946,Z 63,A -98.5307,B 24.8682,C -2.6489,E1 24.994,E2 -538.1099} C_DIS
LIN {X 0.2213,Y -43.1762,Z 63,A -96.113,B 24.8705,C -2.6266,E1 25.0006,E2 -540.4747} C_DIS
Enddeposition()
LIN {X 0.2213,Y -43.1762,Z 63,A -96.113,B 24.8705,C -2.6266,E1 25.0006,E2 -540.4747} C_DIS
Startdeposition()
$VEL.CP = VEL_PRINT
LIN {X -1.3846,Y -42.2098,Z 63,A -99.237,B 24.8702,C -2.629,E1 24.9919,E2 -537.3562} C_DIS
LIN {X -4.2639,Y -42.0169,Z 63,A -103.1901,B 24.8702,C -2.6287,E1 24.9809,E2 -533.4003} C_DIS
LIN {X -7.1714,Y -41.6197,Z 63,A -106.6224,B 24.8694,C -2.6373,E1 24.9715,E2 -529.9856} C_DIS
LIN {X -8.8668,Y -41.2914,Z 63,A -109.211,B 24.8696,C -2.6349,E1 24.9644,E2 -527.3882} C_DIS
LIN {X -11.6646,Y -40.5899,Z 63,A -112.9793,B 24.8692,C -2.6391,E1 24.9542,E2 -523.6244} C_DIS
LIN {X -14.1252,Y -39.8004,Z 63,A -116.5901,B 24.8691,C -2.6404,E1 24.9447,E2 -520.01} C_DIS
LIN {X -16.3747,Y -38.9288,Z 63,A -119.8285,B 24.8687,C -2.644,E1 24.9363,E2 -516.7731} C_DIS
LIN {X -18.639,Y -37.8971,Z 63,A -123.3239,B 24.8685,C -2.6463,E1 24.9274,E2 -513.2742} C_DIS
LIN {X -20.759,Y -36.7788,Z 63,A -126.5757,B 24.8681,C -2.6506,E1 24.9195,E2 -510.0233} C_DIS
LIN {X -22.9139,Y -35.476,Z 63,A -129.999,B 24.8676,C -2.6555,E1 24.9114,E2 -506.6009} C_DIS
LIN {X -25.0196,Y -34.0234,Z 63,A -133.356,B 24.8669,C -2.6626,E1 24.9037,E2 -503.2492} C_DIS
LIN {X -26.8056,Y -32.6345,Z 63,A -136.5252,B 24.8664,C -2.6668,E1 24.8968,E2 -500.0784} C_DIS
LIN {X -28.5416,Y -31.1281,Z 63,A -139.3446,B 24.8655,C -2.6765,E1 24.891,E2 -497.2708} C_DIS
LIN {X -29.6978,Y -30.027,Z 63,A -141.709,B 24.8653,C -2.6784,E1 24.8862,E2 -494.9012} C_DIS
LIN {X -31.0378,Y -28.64,Z 63,A -144.5342,B 24.865,C -2.6815,E1 24.8808,E2 -492.0711} C_DIS
LIN {X -32.8234,Y -26.5745,Z 63,A -147.924,B 24.8637,C -2.6936,E1 24.8747,E2 -488.6945} C_DIS
LIN {X -34.205,Y -24.772,Z 63,A -151.5257,B 24.8637,C -2.6948,E1 24.8687,E2 -485.0785} C_DIS
LIN {X -35.5546,Y -22.7915,Z 63,A -155.0295,B 24.8631,C -2.7001,E1 24.8633,E2 -481.5696} C_DIS
LIN {X -37.2631,Y -19.8765,Z 63,A -159.1636,B 24.8613,C -2.7172,E1 24.8577,E2 -477.4548} C_DIS
LIN {X -38.3491,Y -17.6904,Z 63,A -162.5732,B 24.8605,C -2.7252,E1 24.8536,E2 -474.0458} C_DIS
LIN {X -39.6632,Y -14.5056,Z 63,A -167.0223,B 24.8589,C -2.7409,E1 24.849,E2 -469.6096} C_DIS
LIN {X -40.2448,Y -12.8042,Z 63,A -169.9005,B 24.8587,C -2.7432,E1 24.8465,E2 -466.7202} C_DIS
LIN {X -41.116,Y -9.6477,Z 63,A -173.8895,B 24.8568,C -2.7614,E1 24.8437,E2 -462.7515} C_DIS
LIN {X -41.672,Y -6.8586,Z 63,A -178.6758,B 24.8566,C -2.763,E1 24.8413,E2 -457.9407} C_DIS
LIN {X -42.1433,Y -2.7454,Z 63,A 175.8971,B 24.8546,C -2.7825,E1 24.8399,E2 -452.5277} C_DIS
LIN {X -42.2321,Y 0.1663,Z 63,A 171.8359,B 24.8534,C -2.7937,E1 24.8399,E2 -448.4689} C_DIS
LIN {X -42.0633,Y 3.778,Z 63,A 167.4398,B 24.8512,C -2.8146,E1 24.8406,E2 -444.0963} C_DIS
LIN {X -41.7935,Y 6.0704,Z 63,A 164.406,B 24.85,C -2.8255,E1 24.8417,E2 -441.0704} C_DIS
LIN {X -41.4831,Y 7.9205,Z 63,A 161.2391,B 24.85,C -2.8266,E1 24.8433,E2 -437.8876} C_DIS
LIN {X -40.5274,Y 11.8799,Z 63,A 155.6602,B 24.8481,C -2.8431,E1 24.8473,E2 -432.3156} C_DIS
LIN {X -39.5084,Y 14.9222,Z 63,A 151.7659,B 24.8462,C -2.8612,E1 24.8509,E2 -428.4426} C_DIS
LIN {X -38.6358,Y 17.0547,Z 63,A 148.7116,B 24.8451,C -2.8713,E1 24.8542,E2 -425.3954} C_DIS
LIN {X -37.7992,Y 18.8365,Z 63,A 145.8334,B 24.8445,C -2.8767,E1 24.8577,E2 -422.5147} C_DIS
LIN {X -36.5226,Y 21.2065,Z 63,A 142.6403,B 24.8428,C -2.8922,E1 24.862,E2 -419.3418} C_DIS
LIN {X -35.584,Y 22.7455,Z 63,A 140.0083,B 24.8423,C -2.8969,E1 24.8659,E2 -416.7076} C_DIS
LIN {X -34.6932,Y 24.0824,Z 63,A 137.626,B 24.8419,C -2.9005,E1 24.8696,E2 -414.322} C_DIS
LIN {X -33.3788,Y 25.8738,Z 63,A 134.6974,B 24.841,C -2.9093,E1 24.8745,E2 -411.4006} C_DIS
LIN {X -32.2793,Y 27.2336,Z 63,A 132.3815,B 24.8402,C -2.916,E1 24.8787,E2 -409.0899} C_DIS
LIN {X -30.9113,Y 28.777,Z 63,A 129.2626,B 24.8399,C -2.9192,E1 24.8845,E2 -405.9647} C_DIS
LIN {X -29.1328,Y 30.576,Z 63,A 125.6986,B 24.8392,C -2.9257,E1 24.8916,E2 -402.4013} C_DIS
LIN {X -27.5917,Y 31.9735,Z 63,A 123.2613,B 24.838,C -2.9364,E1 24.8967,E2 -399.9801} C_DIS
LIN {X -26.3393,Y 33.013,Z 63,A 120.4889,B 24.8382,C -2.9344,E1 24.9028,E2 -397.1926} C_DIS
LIN {X -23.7577,Y 34.9159,Z 63,A 116.7093,B 24.8365,C -2.9499,E1 24.9113,E2 -393.4368} C_DIS
LIN {X -22.2298,Y 35.9089,Z 63,A 114.0815,B 24.8362,C -2.9525,E1 24.9175,E2 -390.8069} C_DIS
LIN {X -20.2804,Y 37.0447,Z 63,A 110.8658,B 24.8358,C -2.9559,E1 24.9253,E2 -387.5897} C_DIS
LIN {X -18.4381,Y 37.9953,Z 63,A 108.28,B 24.835,C -2.9631,E1 24.9317,E2 -385.0144} C_DIS
LIN {X -16.319,Y 38.9523,Z 63,A 104.7471,B 24.835,C -2.9629,E1 24.9408,E2 -381.4726} C_DIS
LIN {X -13.8919,Y 39.8824,Z 63,A 101.3385,B 24.8344,C -2.9688,E1 24.9497,E2 -378.0711} C_DIS
LIN {X -11.8018,Y 40.5505,Z 63,A 98.4791,B 24.8338,C -2.9736,E1 24.9573,E2 -375.2183} C_DIS
LIN {X -9.6058,Y 41.1257,Z 63,A 95.1838,B 24.8338,C -2.9736,E1 24.9663,E2 -371.9185} C_DIS
LIN {X -7.0403,Y 41.6415,Z 63,A 91.5368,B 24.8336,C -2.9751,E1 24.9763,E2 -368.2711} C_DIS
LIN {X -4.1377,Y 42.0301,Z 63,A 87.9518,B 24.8328,C -2.9825,E1 24.9862,E2 -364.7015} C_DIS
LIN {X -2.5032,Y 42.1582,Z 63,A 85.6997,B 24.8328,C -2.9831,E1 24.9925,E2 -362.4498} C_DIS
LIN {X -0.4862,Y 42.2297,Z 63,A 82.9476,B 24.8327,C -2.9836,E1 25.0001,E2 -359.6987} C_DIS
LIN {X 2.6524,Y 42.1492,Z 63,A 78.2034,B 24.8334,C -2.9772,E1 25.0134,E2 -354.9405} C_DIS
LIN {X 5.4779,Y 41.8757,Z 63,A 74.7543,B 24.8328,C -2.9822,E1 25.0229,E2 -351.5058} C_DIS
LIN {X 7.5905,Y 41.5449,Z 63,A 71.8163,B 24.833,C -2.9808,E1 25.031,E2 -348.5674} C_DIS
LIN {X 9.4798,Y 41.1548,Z 63,A 68.9143,B 24.8336,C -2.9754,E1 25.039,E2 -345.6565} C_DIS
LIN {X 12.2212,Y 40.4261,Z 63,A 65.2095,B 24.8336,C -2.9749,E1 25.0489,E2 -341.9566} C_DIS
LIN {X 14.429,Y 39.6911,Z 63,A 62.1366,B 24.8338,C -2.9734,E1 25.057,E2 -338.8865} C_DIS
LIN {X 17.0761,Y 38.6269,Z 63,A 57.691,B 24.8353,C -2.9608,E1 25.0685,E2 -334.4214} C_DIS
LIN {X 20.4161,Y 36.9703,Z 63,A 53.5022,B 24.8345,C -2.9676,E1 25.0788,E2 -330.2605} C_DIS
LIN {X 21.7842,Y 36.1809,Z 63,A 51.2724,B 24.835,C -2.9633,E1 25.0842,E2 -328.0271} C_DIS
LIN {X 23.5047,Y 35.0878,Z 63,A 48.807,B 24.835,C -2.9637,E1 25.0899,E2 -325.5708} C_DIS
LIN {X 25.9057,Y 33.3534,Z 63,A 44.4392,B 24.8363,C -2.9514,E1 25.0998,E2 -321.1893} C_DIS
LIN {X 28.0846,Y 31.5412,Z 63,A 40.4543,B 24.8374,C -2.9419,E1 25.1082,E2 -317.1975} C_DIS
LIN {X 30.2091,Y 29.5125,Z 63,A 36.0836,B 24.839,C -2.9275,E1 25.1169,E2 -312.811} C_DIS
LIN {X 32.7041,Y 26.7217,Z 63,A 31.1588,B 24.8399,C -2.9185,E1 25.1259,E2 -307.8874} C_DIS
LIN {X 34.2569,Y 24.7,Z 63,A 27.4974,B 24.8412,C -2.9069,E1 25.1319,E2 -304.216} C_DIS
LIN {X 35.8246,Y 22.3647,Z 63,A 24.0672,B 24.8416,C -2.9036,E1 25.1371,E2 -300.7954} C_DIS
LIN {X 37.1338,Y 20.1163,Z 63,A 20.8445,B 24.842,C -2.8995,E1 25.1415,E2 -297.5796} C_DIS
LIN {X 38.3619,Y 17.6626,Z 63,A 16.6231,B 24.8441,C -2.8809,E1 25.1466,E2 -293.3368} C_DIS
LIN {X 39.39,Y 15.2328,Z 63,A 13.2226,B 24.8448,C -2.8738,E1 25.1501,E2 -289.9383} C_DIS
LIN {X 40.4814,Y 12.0348,Z 63,A 9.0187,B 24.8456,C -2.8669,E1 25.1537,E2 -285.7419} C_DIS
LIN {X 41.1172,Y 9.6426,Z 63,A 5.7215,B 24.8466,C -2.8579,E1 25.156,E2 -282.4425} C_DIS
LIN {X 41.5429,Y 7.6015,Z 63,A 3.0182,B 24.8472,C -2.8514,E1 25.1575,E2 -279.7398} C_DIS
LIN {X 41.916,Y 5.163,Z 63,A -0.2834,B 24.8483,C -2.8419,E1 25.1588,E2 -276.4351} C_DIS
LIN {X 42.0764,Y 3.6249,Z 63,A -2.657,B 24.8495,C -2.8307,E1 25.1594,E2 -274.0488} C_DIS
LIN {X 42.2247,Y 0.8126,Z 63,A -7.0036,B 24.8517,C -2.8097,E1 25.1598,E2 -269.6784} C_DIS
LIN {X 42.1537,Y -2.5753,Z 63,A -10.7393,B 24.8517,C -2.8101,E1 25.1594,E2 -265.9659} C_DIS
LIN {X 41.9509,Y -4.8656,Z 63,A -14.4432,B 24.8538,C -2.7902,E1 25.1583,E2 -262.2368} C_DIS
LIN {X 41.4799,Y -7.9371,Z 63,A -18.3988,B 24.8547,C -2.7815,E1 25.1564,E2 -258.2839} C_DIS
LIN {X 40.8979,Y -10.5331,Z 63,A -21.9256,B 24.8557,C -2.7717,E1 25.1541,E2 -254.7544} C_DIS
LIN {X 40.0765,Y -13.3226,Z 63,A -25.4173,B 24.8561,C -2.7675,E1 25.1513,E2 -251.2725} C_DIS
LIN {X 39.4292,Y -15.1299,Z 63,A -28.2237,B 24.8573,C -2.7561,E1 25.1485,E2 -248.455} C_DIS
LIN {X 38.5886,Y -17.1609,Z 63,A -31.3577,B 24.8585,C -2.7447,E1 25.1451,E2 -245.311} C_DIS
LIN {X 37.7959,Y -18.8431,Z 63,A -33.547,B 24.8587,C -2.743,E1 25.1424,E2 -243.1296} C_DIS
LIN {X 36.6807,Y -20.9314,Z 63,A -37.2844,B 24.8606,C -2.7249,E1 25.1373,E2 -239.3687} C_DIS
LIN {X 35.552,Y -22.7955,Z 63,A -40.6599,B 24.8621,C -2.7096,E1 25.1322,E2 -235.9742} C_DIS
LIN {X 32.8968,Y -26.484,Z 63,A -46.0907,B 24.8625,C -2.7057,E1 25.1232,E2 -230.5599} C_DIS
LIN {X 30.7971,Y -28.8985,Z 63,A -50.6506,B 24.864,C -2.6913,E1 25.1146,E2 -225.9862} C_DIS
LIN {X 29.0477,Y -30.6568,Z 63,A -53.5251,B 24.864,C -2.6915,E1 25.1089,E2 -223.1242} C_DIS
LIN {X 27.2091,Y -32.2989,Z 63,A -57.5235,B 24.8658,C -2.6733,E1 25.1004,E2 -219.0985} C_DIS
LIN {X 24.7316,Y -34.2344,Z 63,A -61.8967,B 24.8669,C -2.6628,E1 25.0906,E2 -214.716} C_DIS
LIN {X 21.5336,Y -36.3302,Z 63,A -66.0566,B 24.8662,C -2.6696,E1 25.0808,E2 -210.5857} C_DIS
LIN {X 19.3131,Y -37.5579,Z 63,A -70.2097,B 24.8679,C -2.6525,E1 25.0705,E2 -206.4039} C_DIS
LIN {X 16.8825,Y -38.7113,Z 63,A -73.2562,B 24.8675,C -2.6565,E1 25.0629,E2 -203.3745} C_DIS
LIN {X 13.9261,Y -39.8704,Z 63,A -78.6415,B 24.8697,C -2.6342,E1 25.0486,E2 -197.9478} C_DIS
LIN {X 11.3392,Y -40.6821,Z 63,A -81.824,B 24.8694,C -2.6378,E1 25.0402,E2 -194.7789} C_DIS
LIN {X 8.5861,Y -41.3506,Z 63,A -85.3824,B 24.8693,C -2.6386,E1 25.0305,E2 -191.2272} C_DIS
LIN {X 5.8267,Y -41.8287,Z 63,A -89.0302,B 24.8693,C -2.6381,E1 25.0204,E2 -187.5819} C_DIS
Enddeposition()
END
